C03635=1018.441,60.715,389.816,166.714,53.558,159.792
C03636=1018.447,60.965,389.800,166.716,53.550,159.791
C03637=1018.453,61.215,389.784,166.719,53.543,159.790
C03638=1018.458,61.464,389.769,166.722,53.536,159.789
C03639=1018.463,61.714,389.752,166.725,53.528,159.788
C03640=1018.469,61.964,389.737,166.727,53.521,159.787
C03641=1018.474,62.213,389.720,166.730,53.514,159.786
C03642=1018.480,62.462,389.704,166.732,53.506,159.785
C03643=1018.485,62.712,389.689,166.735,53.499,159.784
C03644=1018.491,62.961,389.673,166.738,53.491,159.784
C03645=1018.496,63.211,389.657,166.740,53.485,159.783
C03646=1018.502,63.460,389.641,166.743,53.477,159.782
C03647=1018.507,63.701,389.624,166.745,53.470,159.781
C03648=1018.512,63.942,389.609,166.748,53.463,159.780
C03649=1018.518,64.183,389.593,166.750,53.456,159.779
C03650=1018.523,64.424,389.578,166.753,53.449,159.779
C03651=1018.528,64.666,389.562,166.756,53.442,159.778
C03652=1018.533,64.907,389.546,166.758,53.435,159.777
C03653=1018.539,65.148,389.531,166.761,53.428,159.776
C03654=1018.543,65.389,389.515,166.763,53.421,159.775
C03655=1018.549,65.638,389.499,166.766,53.414,159.774
C03656=1018.554,65.888,389.482,166.768,53.407,159.773
C03657=1018.560,66.137,389.466,166.770,53.399,159.772
C03658=1018.565,66.387,389.450,166.773,53.392,159.772
C03659=1018.571,66.636,389.434,166.777,53.385,159.771
C03660=1018.576,66.885,389.418,166.778,53.378,159.770
C03661=1018.581,67.135,389.401,166.781,53.371,159.769
C03662=1018.587,67.384,389.385,166.785,53.363,159.768
C03663=1018.592,67.634,389.369,166.786,53.356,159.767
C03664=1018.597,67.883,389.353,166.789,53.349,159.766
C03665=1018.603,68.133,389.336,166.792,53.342,159.766
C03666=1018.609,68.382,389.320,166.795,53.334,159.765
C03667=1018.614,68.632,389.303,166.797,53.327,159.764
C03668=1018.619,68.880,389.287,166.800,53.320,159.763
C03669=1018.624,69.130,389.270,166.803,53.312,159.762
C03670=1018.630,69.380,389.253,166.805,53.306,159.761
C03671=1018.635,69.629,389.237,166.808,53.298,159.761
C03672=1018.640,69.878,389.221,166.811,53.291,159.760
C03673=1018.646,70.127,389.204,166.813,53.284,159.759
C03674=1018.651,70.377,389.187,166.816,53.277,159.758
C03675=1018.656,70.627,389.171,166.818,53.269,159.757
C03676=1018.662,70.876,389.154,166.820,53.262,159.756
C03677=1018.667,71.125,389.138,166.823,53.255,159.755
C03678=1018.673,71.374,389.122,166.826,53.248,159.755
C03679=1018.678,71.624,389.105,166.828,53.241,159.754
C03680=1018.683,71.874,389.088,166.831,53.234,159.753
C03681=1018.689,72.123,389.072,166.834,53.226,159.752
C03682=1018.694,72.372,389.055,166.836,53.219,159.751
C03683=1018.699,72.621,389.038,166.839,53.212,159.750
C03684=1018.705,72.871,389.022,166.842,53.205,159.749
C03685=1018.710,73.120,389.005,166.845,53.198,159.749
C03686=1018.716,73.370,388.988,166.847,53.190,159.747
C03687=1018.721,73.619,388.972,166.850,53.183,159.747
C03688=1018.726,73.868,388.956,166.853,53.176,159.746
C03689=1018.732,74.118,388.939,166.855,53.169,159.745
C03690=1018.737,74.367,388.922,166.858,53.162,159.744
C03691=1018.743,74.666,388.902,166.861,53.153,159.743
C03692=1018.750,74.965,388.882,166.864,53.144,159.742
C03693=1018.756,75.265,388.862,166.868,53.136,159.741
C03694=1018.763,75.563,388.842,166.871,53.127,159.740
C03695=1018.768,75.813,388.825,166.873,53.120,159.739
C03696=1018.774,76.062,388.809,166.876,53.112,159.738
C03697=1018.780,76.312,388.792,166.879,53.105,159.737
C03698=1018.785,76.560,388.775,166.881,53.098,159.736
C03699=1018.790,76.810,388.758,166.884,53.091,159.736
C03700=1018.796,77.059,388.742,166.887,53.084,159.735
C03701=1018.801,77.309,388.725,166.888,53.076,159.734
C03702=1018.806,77.559,388.708,166.891,53.069,159.733
C03703=1018.812,77.808,388.691,166.894,53.062,159.732
C03704=1018.817,78.057,388.674,166.897,53.055,159.731
C03705=1018.822,78.307,388.657,166.900,53.048,159.730
C03706=1018.828,78.556,388.640,166.903,53.041,159.730
C03707=1018.832,78.805,388.623,166.905,53.034,159.729
C03708=1018.837,79.055,388.606,166.908,53.027,159.728
C03709=1018.843,79.304,388.589,166.910,53.019,159.727
C03710=1018.848,79.553,388.572,166.912,53.012,159.726
C03711=1018.854,79.803,388.556,166.915,53.005,159.725
C03712=1018.860,80.052,388.538,166.919,52.998,159.725
C03713=1018.865,80.301,388.521,166.921,52.991,159.724
C03714=1018.870,80.551,388.504,166.924,52.984,159.723
C03715=1018.876,80.800,388.487,166.927,52.977,159.722
C03716=1018.881,81.050,388.470,166.928,52.969,159.721
C03717=1018.886,81.299,388.453,166.931,52.962,159.720
C03718=1018.891,81.548,388.436,166.934,52.955,159.719
C03719=1018.896,81.797,388.419,166.937,52.948,159.718
C03720=1018.902,82.046,388.401,166.940,52.941,159.718
C03721=1018.907,82.296,388.385,166.942,52.933,159.717
C03722=1018.912,82.546,388.368,166.944,52.927,159.716
C03723=1018.918,82.795,388.350,166.947,52.919,159.715
C03724=1018.923,83.044,388.333,166.950,52.912,159.714
C03725=1018.928,83.293,388.316,166.953,52.905,159.713
C03726=1018.934,83.543,388.299,166.955,52.898,159.712
C03727=1018.939,83.792,388.283,166.958,52.890,159.712
C03728=1018.945,84.041,388.265,166.961,52.883,159.711
C03729=1018.950,84.291,388.248,166.963,52.877,159.710
C03730=1018.956,84.540,388.231,166.966,52.869,159.709
C03731=1018.961,84.790,388.214,166.969,52.862,159.708
C03732=1018.966,85.039,388.196,166.971,52.855,159.707
C03733=1018.972,85.289,388.179,166.974,52.848,159.706
C03734=1018.977,85.538,388.162,166.977,52.840,159.705
C03735=1018.982,85.787,388.145,166.980,52.833,159.705
C03736=1018.988,86.036,388.127,166.982,52.826,159.704
C03737=1018.993,86.286,388.110,166.985,52.819,159.703
C03738=1018.998,86.536,388.094,166.988,52.811,159.702
C03739=1019.004,86.785,388.076,166.990,52.804,159.701
C03740=1019.009,87.034,388.059,166.993,52.797,159.700
C03741=1019.015,87.283,388.042,166.996,52.789,159.699
C03742=1019.020,87.532,388.024,166.999,52.782,159.698
C03743=1019.025,87.782,388.007,167.001,52.775,159.698
C03744=1019.032,88.031,387.990,167.004,52.768,159.697
C03745=1019.037,88.280,387.973,167.007,52.760,159.696
C03746=1019.042,88.529,387.956,167.010,52.753,159.695
C03747=1019.048,88.779,387.939,167.012,52.747,159.694
C03748=1019.053,89.028,387.921,167.015,52.739,159.693
C03749=1019.058,89.278,387.904,167.018,52.732,159.692
C03750=1019.064,89.528,387.886,167.021,52.725,159.692
C03751=1019.069,89.777,387.868,167.023,52.718,159.691
C03752=1019.074,90.027,387.852,167.026,52.711,159.690
C03753=1019.079,90.276,387.833,167.029,52.703,159.689
C03754=1019.085,90.525,387.816,167.031,52.696,159.688
C03755=1019.091,90.807,387.796,167.034,52.688,159.687
C03756=1019.097,91.090,387.776,167.037,52.680,159.686
C03757=1019.102,91.373,387.756,167.040,52.672,159.685
C03758=1019.108,91.654,387.737,167.044,52.664,159.684
C03759=1019.115,91.904,387.719,167.047,52.657,159.683
C03760=1019.119,92.154,387.701,167.048,52.650,159.682
C03761=1019.125,92.403,387.683,167.051,52.642,159.682
C03762=1019.130,92.652,387.667,167.055,52.635,159.681
C03763=1019.135,92.902,387.648,167.057,52.629,159.680
C03764=1019.140,93.151,387.631,167.060,52.622,159.679
C03765=1019.146,93.400,387.613,167.063,52.614,159.678
C03766=1019.151,93.649,387.596,167.065,52.607,159.677
C03767=1019.156,93.899,387.578,167.068,52.600,159.676
C03768=1019.161,94.148,387.561,167.071,52.593,159.676
C03769=1019.167,94.397,387.543,167.074,52.585,159.675
C03770=1019.173,94.646,387.525,167.076,52.578,159.674
C03771=1019.178,94.896,387.507,167.079,52.571,159.673
C03772=1019.183,95.145,387.490,167.082,52.564,159.672
C03773=1019.188,95.395,387.473,167.084,52.557,159.671
C03774=1019.194,95.644,387.455,167.087,52.550,159.670
C03775=1019.199,95.893,387.437,167.090,52.542,159.669
C03776=1019.204,96.142,387.419,167.093,52.535,159.669
C03777=1019.210,96.392,387.401,167.095,52.528,159.668
C03778=1019.215,96.641,387.383,167.098,52.521,159.667
C03779=1019.221,96.890,387.366,167.101,52.514,159.666
C03780=1019.226,97.140,387.349,167.104,52.507,159.665
C03781=1019.231,97.389,387.331,167.106,52.499,159.664
C03782=1019.236,97.638,387.313,167.109,52.492,159.663
C03783=1019.242,97.888,387.295,167.112,52.485,159.663
C03784=1019.248,98.137,387.278,167.115,52.477,159.662
C03785=1019.253,98.386,387.260,167.117,52.471,159.661
C03786=1019.258,98.635,387.242,167.120,52.464,159.660
C03787=1019.264,98.884,387.224,167.123,52.456,159.659
C03788=1019.270,99.134,387.206,167.126,52.449,159.658
C03789=1019.275,99.383,387.188,167.128,52.442,159.657
C03790=1019.280,99.632,387.171,167.131,52.435,159.656
C03791=1019.285,99.882,387.152,167.135,52.428,159.656
C03792=1019.290,100.131,387.135,167.137,52.421,159.655
C03793=1019.296,100.381,387.116,167.139,52.413,159.654
C03794=1019.301,100.630,387.098,167.143,52.406,159.653
C03795=1019.306,100.879,387.081,167.145,52.400,159.652
C03796=1019.311,101.129,387.062,167.148,52.393,159.651
C03797=1019.316,101.378,387.045,167.151,52.385,159.651
C03798=1019.322,101.627,387.026,167.153,52.378,159.649
C03799=1019.328,101.876,387.008,167.156,52.371,159.649
C03800=1019.332,102.126,386.990,167.159,52.364,159.648
C03801=1019.337,102.375,386.972,167.162,52.357,159.647
C03802=1019.343,102.625,386.954,167.164,52.350,159.646
C03803=1019.348,102.874,386.936,167.168,52.343,159.645
C03804=1019.354,103.123,386.918,167.170,52.335,159.644
C03805=1019.359,103.372,386.899,167.172,52.329,159.643
C03806=1019.365,103.621,386.881,167.176,52.322,159.643
C03807=1019.370,103.871,386.863,167.179,52.315,159.642
C03808=1019.374,104.120,386.845,167.182,52.307,159.641
C03809=1019.380,104.369,386.827,167.184,52.300,159.640
C03810=1019.385,104.619,386.809,167.187,52.293,159.639
C03811=1019.391,104.868,386.791,167.190,52.286,159.638
C03812=1019.396,105.117,386.772,167.192,52.279,159.637
C03813=1019.401,105.366,386.755,167.195,52.272,159.637
C03814=1019.407,105.616,386.736,167.198,52.264,159.636
C03815=1019.412,105.865,386.717,167.201,52.257,159.635
C03816=1019.417,106.114,386.700,167.203,52.250,159.634
C03817=1019.423,106.364,386.681,167.206,52.243,159.633
C03818=1019.428,106.613,386.664,167.209,52.236,159.632
C03819=1019.434,106.895,386.643,167.212,52.228,159.631
C03820=1019.441,107.178,386.622,167.216,52.219,159.630
C03821=1019.447,107.461,386.602,167.219,52.211,159.629
C03822=1019.453,107.743,386.581,167.222,52.204,159.628
C03823=1019.458,107.993,386.562,167.225,52.197,159.628
C03824=1019.463,108.242,386.544,167.228,52.189,159.627
C03825=1019.468,108.491,386.527,167.230,52.182,159.626
C03826=1019.474,108.741,386.507,167.234,52.175,159.625
C03827=1019.480,108.990,386.490,167.236,52.167,159.624
C03828=1019.484,109.239,386.472,167.239,52.160,159.623
C03829=1019.491,109.488,386.453,167.243,52.153,159.622
C03830=1019.495,109.737,386.435,167.245,52.147,159.622
C03831=1019.500,109.987,386.417,167.248,52.139,159.621
C03832=1019.506,110.236,386.397,167.251,52.132,159.620
C03833=1019.511,110.486,386.379,167.254,52.125,159.619
C03834=1019.517,110.734,386.361,167.256,52.118,159.618
C03835=1019.522,110.984,386.342,167.259,52.110,159.617
C03836=1019.527,111.233,386.324,167.262,52.103,159.616
C03837=1019.532,111.482,386.305,167.265,52.096,159.616
C03838=1019.538,111.732,386.287,167.268,52.090,159.615
C03839=1019.543,111.981,386.269,167.270,52.082,159.614
C03840=1019.548,112.231,386.250,167.274,52.075,159.613
C03841=1019.553,112.479,386.231,167.277,52.068,159.612
C03842=1019.558,112.729,386.213,167.279,52.061,159.611
C03843=1019.564,112.978,386.194,167.282,52.054,159.610
C03844=1019.569,113.227,386.175,167.285,52.047,159.610
C03845=1019.574,113.477,386.156,167.288,52.041,159.609
C03846=1019.580,113.726,386.137,167.291,52.034,159.608
C03847=1019.585,113.974,386.119,167.294,52.027,159.607
C03848=1019.590,114.224,386.100,167.296,52.019,159.606
C03849=1019.595,114.473,386.081,167.299,52.012,159.605
C03850=1019.600,114.722,386.062,167.302,52.005,159.605
C03851=1019.606,114.972,386.044,167.305,51.999,159.604
C03852=1019.611,115.221,386.025,167.308,51.992,159.603
C03853=1019.616,115.470,386.005,167.311,51.985,159.602
C03854=1019.620,115.720,385.987,167.314,51.978,159.601
C03855=1019.625,115.968,385.968,167.316,51.971,159.600
C03856=1019.631,116.218,385.949,167.319,51.963,159.599
C03857=1019.636,116.467,385.931,167.322,51.956,159.599
C03858=1019.642,116.717,385.911,167.325,51.950,159.598
C03859=1019.647,116.965,385.893,167.328,51.943,159.597
C03860=1019.652,117.215,385.874,167.331,51.936,159.596
C03861=1019.657,117.464,385.855,167.334,51.929,159.595
C03862=1019.663,117.714,385.836,167.336,51.921,159.594
C03863=1019.668,117.962,385.817,167.339,51.914,159.594
C03864=1019.673,118.212,385.799,167.343,51.907,159.593
C03865=1019.678,118.461,385.780,167.346,51.900,159.592
C03866=1019.683,118.710,385.761,167.348,51.894,159.591
C03867=1019.689,118.959,385.741,167.351,51.887,159.590
C03868=1019.694,119.209,385.723,167.354,51.879,159.589
C03869=1019.699,119.458,385.703,167.357,51.872,159.589
C03870=1019.704,119.707,385.685,167.360,51.865,159.588
C03871=1019.710,119.957,385.665,167.363,51.858,159.587
C03872=1019.715,120.205,385.646,167.366,51.851,159.586
C03873=1019.720,120.455,385.628,167.369,51.844,159.585
C03874=1019.725,120.704,385.609,167.372,51.837,159.584
C03875=1019.731,120.954,385.590,167.374,51.830,159.583
C03876=1019.736,121.202,385.571,167.378,51.823,159.583
C03877=1019.742,121.452,385.552,167.381,51.815,159.582
C03878=1019.747,121.700,385.533,167.384,51.808,159.581
C03879=1019.752,121.950,385.514,167.387,51.801,159.580
C03880=1019.757,122.199,385.495,167.389,51.795,159.579
C03881=1019.763,122.449,385.476,167.393,51.788,159.578
C03882=1019.768,122.697,385.457,167.395,51.780,159.577
C03883=1019.774,122.980,385.435,167.399,51.772,159.577
C03884=1019.780,123.263,385.413,167.402,51.764,159.576
C03885=1019.786,123.545,385.392,167.406,51.756,159.575
C03886=1019.792,123.828,385.370,167.408,51.748,159.574
C03887=1019.798,124.078,385.351,167.412,51.741,159.573
C03888=1019.803,124.326,385.332,167.415,51.734,159.572
C03889=1019.808,124.576,385.313,167.418,51.727,159.571
C03890=1019.814,124.824,385.294,167.421,51.719,159.570
C03891=1019.819,125.074,385.276,167.424,51.713,159.569
C03892=1019.824,125.323,385.257,167.427,51.706,159.569
C03893=1019.830,125.573,385.238,167.430,51.698,159.568
C03894=1019.835,125.822,385.218,167.433,51.691,159.567
C03895=1019.840,126.071,385.199,167.436,51.684,159.566
C03896=1019.845,126.321,385.180,167.439,51.677,159.565
C03897=1019.850,126.569,385.161,167.442,51.670,159.564
C03898=1019.856,126.819,385.141,167.445,51.663,159.563
C03899=1019.862,127.068,385.122,167.449,51.656,159.563
C03900=1019.867,127.317,385.103,167.451,51.648,159.562
C03901=1019.873,127.566,385.084,167.454,51.642,159.561
C03902=1019.878,127.816,385.065,167.457,51.635,159.560
C03903=1019.883,128.064,385.046,167.460,51.627,159.559
C03904=1019.889,128.314,385.027,167.463,51.620,159.558
C03905=1019.894,128.564,385.007,167.467,51.613,159.557
C03906=1019.899,128.812,384.988,167.469,51.605,159.557
C03907=1019.905,129.062,384.969,167.473,51.598,159.556
C03908=1019.910,129.311,384.950,167.476,51.592,159.555
C03909=1019.916,129.560,384.931,167.479,51.584,159.554
C03910=1019.921,129.809,384.911,167.482,51.577,159.553
C03911=1019.927,130.059,384.892,167.485,51.570,159.552
C03912=1019.932,130.307,384.872,167.488,51.563,159.552
C03913=1019.937,130.557,384.853,167.491,51.556,159.551
C03914=1019.942,130.806,384.833,167.494,51.549,159.550
C03915=1019.947,131.055,384.814,167.497,51.542,159.549
C03916=1019.952,131.305,384.794,167.500,51.535,159.548
C03917=1019.958,131.554,384.774,167.503,51.528,159.547
C03918=1019.963,131.803,384.755,167.506,51.521,159.547
C03919=1019.968,132.052,384.736,167.509,51.514,159.546
C03920=1019.974,132.301,384.716,167.512,51.507,159.545
C03921=1019.979,132.550,384.696,167.516,51.500,159.544
C03922=1019.984,132.799,384.677,167.519,51.493,159.543
C03923=1019.989,133.049,384.657,167.521,51.486,159.542
C03924=1019.995,133.297,384.637,167.524,51.479,159.541
C03925=1020.000,133.547,384.618,167.527,51.472,159.541
C03926=1020.005,133.797,384.598,167.531,51.465,159.540
C03927=1020.011,134.045,384.578,167.534,51.458,159.539
C03928=1020.016,134.294,384.559,167.537,51.451,159.538
C03929=1020.021,134.544,384.540,167.540,51.443,159.537
C03930=1020.027,134.793,384.519,167.543,51.437,159.536
C03931=1020.032,135.042,384.500,167.546,51.430,159.536
C03932=1020.037,135.291,384.480,167.549,51.423,159.535
C03933=1020.043,135.540,384.460,167.553,51.416,159.534
C03934=1020.048,135.790,384.441,167.555,51.409,159.533
C03935=1020.053,136.039,384.422,167.559,51.402,159.532
C03936=1020.058,136.288,384.401,167.562,51.395,159.531
C03937=1020.064,136.537,384.382,167.565,51.388,159.531
C03938=1020.069,136.786,384.361,167.569,51.381,159.530
C03939=1020.074,137.035,384.342,167.571,51.374,159.529
C03940=1020.079,137.284,384.322,167.574,51.367,159.528
C03941=1020.085,137.534,384.303,167.577,51.360,159.527
C03942=1020.090,137.783,384.282,167.581,51.353,159.527
C03943=1020.096,138.032,384.263,167.584,51.346,159.526
C03944=1020.100,138.281,384.243,167.587,51.338,159.525
C03945=1020.105,138.530,384.223,167.590,51.331,159.524
C03946=1020.111,138.780,384.202,167.593,51.325,159.523
C03947=1020.117,139.062,384.180,167.596,51.317,159.522
C03948=1020.123,139.345,384.158,167.600,51.309,159.521
C03949=1020.129,139.627,384.135,167.604,51.301,159.520
C03950=1020.135,139.910,384.112,167.607,51.293,159.519
C03951=1020.140,140.158,384.093,167.611,51.287,159.519
C03952=1020.145,140.408,384.072,167.614,51.280,159.518
C03953=1020.150,140.657,384.052,167.617,51.273,159.517
C03954=1020.155,140.906,384.032,167.620,51.265,159.516
C03955=1020.161,141.155,384.012,167.624,51.258,159.515
C03956=1020.166,141.404,383.992,167.627,51.251,159.515
C03957=1020.171,141.653,383.972,167.630,51.245,159.514
C03958=1020.177,141.902,383.952,167.634,51.238,159.513
C03959=1020.182,142.152,383.932,167.636,51.231,159.512
C03960=1020.187,142.401,383.912,167.639,51.224,159.511
C03961=1020.192,142.650,383.891,167.642,51.217,159.510
C03962=1020.197,142.899,383.872,167.646,51.210,159.510
C03963=1020.203,143.148,383.852,167.649,51.203,159.509
C03964=1020.208,143.397,383.831,167.652,51.196,159.508
C03965=1020.214,143.646,383.811,167.656,51.189,159.507
C03966=1020.219,143.896,383.791,167.659,51.182,159.506
C03967=1020.224,144.145,383.771,167.662,51.175,159.506
C03968=1020.229,144.394,383.750,167.665,51.168,159.505
C03969=1020.235,144.643,383.731,167.669,51.161,159.504
C03970=1020.240,144.893,383.710,167.672,51.154,159.503
C03971=1020.245,145.141,383.690,167.675,51.147,159.502
C03972=1020.251,145.390,383.670,167.678,51.140,159.501
C03973=1020.256,145.640,383.650,167.682,51.133,159.501
C03974=1020.261,145.889,383.630,167.685,51.126,159.500
C03975=1020.266,146.138,383.609,167.688,51.119,159.499
C03976=1020.272,146.387,383.589,167.692,51.112,159.498
C03977=1020.277,146.636,383.568,167.695,51.105,159.498
C03978=1020.282,146.885,383.548,167.697,51.099,159.497
C03979=1020.288,147.134,383.528,167.700,51.091,159.496
C03980=1020.293,147.384,383.508,167.704,51.084,159.495
C03981=1020.298,147.633,383.487,167.707,51.077,159.494
C03982=1020.304,147.882,383.467,167.710,51.071,159.493
C03983=1020.309,148.131,383.446,167.714,51.064,159.493
C03984=1020.314,148.379,383.426,167.717,51.057,159.492
C03985=1020.319,148.629,383.405,167.721,51.050,159.491
C03986=1020.324,148.878,383.385,167.724,51.043,159.490
C03987=1020.329,149.127,383.364,167.727,51.036,159.489
C03988=1020.335,149.376,383.344,167.731,51.029,159.489
C03989=1020.340,149.625,383.323,167.734,51.022,159.488
C03990=1020.345,149.874,383.303,167.737,51.016,159.487
C03991=1020.350,150.123,383.282,167.740,51.008,159.486
C03992=1020.356,150.372,383.261,167.744,51.001,159.485
C03993=1020.361,150.622,383.241,167.747,50.994,159.485
C03994=1020.366,150.871,383.220,167.751,50.988,159.484
C03995=1020.371,151.120,383.200,167.754,50.981,159.483
C03996=1020.377,151.369,383.179,167.757,50.974,159.482
C03997=1020.382,151.618,383.159,167.761,50.967,159.481
C03998=1020.387,151.867,383.138,167.764,50.960,159.481
C03999=1020.392,152.116,383.118,167.767,50.953,159.480
C04000=1020.398,152.365,383.097,167.771,50.946,159.479
C04001=1020.403,152.614,383.076,167.774,50.939,159.478
C04002=1020.408,152.863,383.055,167.777,50.932,159.477
C04003=1020.414,153.112,383.035,167.781,50.925,159.477
C04004=1020.419,153.361,383.014,167.784,50.918,159.476
C04005=1020.424,153.610,382.994,167.787,50.912,159.475
C04006=1020.429,153.860,382.972,167.791,50.905,159.474
C04007=1020.434,154.109,382.952,167.794,50.898,159.473
C04008=1020.440,154.358,382.930,167.798,50.891,159.473
C04009=1020.445,154.607,382.910,167.801,50.884,159.472
C04010=1020.451,154.857,382.889,167.804,50.877,159.471
C04011=1020.456,155.139,382.865,167.807,50.870,159.470
C04012=1020.462,155.421,382.842,167.811,50.862,159.469
C04013=1020.469,155.703,382.818,167.815,50.854,159.468
C04014=1020.474,155.985,382.795,167.819,50.846,159.467
C04015=1020.480,156.234,382.774,167.823,50.839,159.467
C04016=1020.484,156.483,382.753,167.826,50.833,159.466
C04017=1020.490,156.733,382.732,167.830,50.826,159.465
C04018=1020.495,156.982,382.711,167.833,50.819,159.464
C04019=1020.501,157.231,382.690,167.837,50.812,159.464
C04020=1020.506,157.480,382.670,167.840,50.805,159.463
C04021=1020.511,157.729,382.649,167.843,50.799,159.462
C04022=1020.516,157.978,382.627,167.847,50.792,159.461
C04023=1020.521,158.227,382.607,167.850,50.785,159.460
C04024=1020.527,158.476,382.586,167.853,50.777,159.459
C04025=1020.532,158.725,382.565,167.857,50.771,159.459
C04026=1020.538,158.974,382.544,167.860,50.764,159.458
C04027=1020.543,159.223,382.522,167.864,50.758,159.457
C04028=1020.547,159.473,382.501,167.867,50.751,159.457
C04029=1020.553,159.721,382.480,167.871,50.744,159.456
C04030=1020.558,159.971,382.458,167.874,50.737,159.455
C04031=1020.563,160.219,382.437,167.877,50.730,159.454
C04032=1020.568,160.468,382.415,167.881,50.724,159.453
C04033=1020.572,160.717,382.394,167.885,50.717,159.453
C04034=1020.579,160.967,382.372,167.888,50.711,159.452
C04035=1020.583,161.216,382.351,167.892,50.704,159.451
C04036=1020.588,161.465,382.329,167.895,50.697,159.451
C04037=1020.593,161.713,382.308,167.898,50.690,159.450
C04038=1020.598,161.963,382.287,167.902,50.683,159.449
C04039=1020.604,162.211,382.266,167.906,50.677,159.448
C04040=1020.608,162.460,382.244,167.909,50.671,159.448
C04041=1020.614,162.710,382.222,167.912,50.664,159.447
C04042=1020.619,162.959,382.201,167.916,50.657,159.446
C04043=1020.624,163.208,382.179,167.919,50.650,159.445
C04044=1020.628,163.457,382.158,167.923,50.643,159.444
C04045=1020.634,163.706,382.137,167.927,50.637,159.444
C04046=1020.639,163.954,382.115,167.930,50.630,159.443
C04047=1020.645,164.204,382.094,167.933,50.624,159.442
C04048=1020.649,164.453,382.072,167.937,50.617,159.442
C04049=1020.654,164.702,382.050,167.940,50.610,159.441
C04050=1020.660,164.950,382.029,167.944,50.603,159.440
C04051=1020.665,165.200,382.008,167.947,50.597,159.439
C04052=1020.670,165.449,381.986,167.951,50.590,159.439
C04053=1020.675,165.698,381.964,167.954,50.584,159.438
C04054=1020.680,165.947,381.943,167.958,50.577,159.437
C04055=1020.685,166.197,381.921,167.961,50.570,159.436
C04056=1020.691,166.445,381.900,167.965,50.563,159.435
C04057=1020.696,166.694,381.878,167.969,50.556,159.435
C04058=1020.701,166.943,381.857,167.973,50.549,159.434
C04059=1020.707,167.192,381.834,167.977,50.543,159.433
C04060=1020.711,167.441,381.813,167.980,50.537,159.433
C04061=1020.717,167.690,381.792,167.983,50.530,159.432
C04062=1020.722,167.939,381.770,167.987,50.523,159.431
C04063=1020.727,168.188,381.748,167.990,50.516,159.430
C04064=1020.733,168.437,381.727,167.994,50.509,159.430
C04065=1020.737,168.686,381.705,167.997,50.503,159.429
C04066=1020.743,168.936,381.683,168.001,50.496,159.428
C04067=1020.748,169.184,381.662,168.005,50.490,159.427
C04068=1020.753,169.433,381.640,168.009,50.483,159.427
C04069=1020.759,169.682,381.618,168.012,50.476,159.426
C04070=1020.764,169.931,381.597,168.016,50.469,159.425
C04071=1020.769,170.180,381.575,168.019,50.462,159.424
C04072=1020.775,170.429,381.553,168.023,50.456,159.424
C04073=1020.780,170.678,381.531,168.026,50.449,159.423
C04074=1020.785,170.927,381.509,168.030,50.442,159.422
C04075=1020.791,171.209,381.485,168.034,50.435,159.421
C04076=1020.797,171.491,381.460,168.038,50.427,159.420
C04077=1020.803,171.773,381.436,168.042,50.420,159.420
C04078=1020.809,172.055,381.411,168.047,50.412,159.419
C04079=1020.814,172.304,381.389,168.050,50.405,159.418
C04080=1020.819,172.553,381.368,168.055,50.399,159.417
C04081=1020.825,172.802,381.345,168.058,50.392,159.417
C04082=1020.830,173.051,381.324,168.062,50.385,159.416
C04083=1020.836,173.300,381.302,168.065,50.378,159.415
C04084=1020.841,173.549,381.280,168.069,50.372,159.414
C04085=1020.847,173.798,381.258,168.073,50.365,159.414
C04086=1020.851,174.047,381.236,168.077,50.358,159.413
C04087=1020.856,174.296,381.215,168.080,50.351,159.412
C04088=1020.862,174.545,381.193,168.084,50.344,159.411
C04089=1020.867,174.794,381.171,168.087,50.338,159.411
C04090=1020.873,175.043,381.149,168.092,50.331,159.410
C04091=1020.878,175.292,381.128,168.095,50.324,159.409
C04092=1020.884,175.541,381.105,168.099,50.318,159.408
C04093=1020.889,175.790,381.083,168.102,50.311,159.408
C04094=1020.895,176.039,381.061,168.107,50.304,159.407
C04095=1020.900,176.288,381.039,168.110,50.297,159.406
C04096=1020.905,176.537,381.017,168.114,50.290,159.405
C04097=1020.911,176.786,380.996,168.117,50.284,159.405
C04098=1020.916,177.035,380.974,168.122,50.277,159.404
C04099=1020.921,177.284,380.952,168.126,50.271,159.403
C04100=1020.928,177.532,380.929,168.129,50.264,159.402
C04101=1020.932,177.781,380.907,168.133,50.257,159.402
C04102=1020.938,178.031,380.885,168.137,50.250,159.401
C04103=1020.943,178.279,380.864,168.141,50.243,159.400
C04104=1020.949,178.529,380.842,168.144,50.237,159.399
C04105=1020.954,178.777,380.819,168.149,50.230,159.399
C04106=1020.960,179.026,380.798,168.153,50.223,159.398
C04107=1020.965,179.275,380.776,168.156,50.217,159.397
C04108=1020.970,179.525,380.753,168.161,50.210,159.397
C04109=1020.976,179.774,380.732,168.164,50.203,159.396
C04110=1020.982,180.022,380.709,168.168,50.196,159.395
C04111=1020.987,180.271,380.687,168.172,50.189,159.394
C04112=1020.993,180.520,380.666,168.176,50.183,159.394
C04113=1020.998,180.769,380.643,168.179,50.176,159.393
C04114=1021.004,181.018,380.621,168.183,50.169,159.392
C04115=1021.009,181.267,380.599,168.187,50.163,159.392
C04116=1021.015,181.516,380.577,168.191,50.156,159.391
C04117=1021.020,181.765,380.554,168.195,50.149,159.390
C04118=1021.025,182.014,380.532,168.199,50.142,159.389
C04119=1021.032,182.263,380.510,168.202,50.136,159.389
C04120=1021.036,182.512,380.487,168.206,50.130,159.388
C04121=1021.042,182.761,380.464,168.211,50.123,159.387
C04122=1021.046,183.011,380.442,168.215,50.116,159.387
C04123=1021.051,183.259,380.419,168.218,50.110,159.386
C04124=1021.057,183.508,380.396,168.222,50.103,159.385
C04125=1021.062,183.756,380.374,168.226,50.097,159.384
C04126=1021.067,184.006,380.351,168.230,50.090,159.384
C04127=1021.073,184.255,380.328,168.234,50.084,159.383
C04128=1021.077,184.503,380.306,168.238,50.077,159.382
C04129=1021.082,184.753,380.282,168.241,50.071,159.382
C04130=1021.088,185.002,380.259,168.245,50.065,159.381
C04131=1021.093,185.250,380.238,168.250,50.058,159.381
C04132=1021.098,185.500,380.214,168.253,50.052,159.380
C04133=1021.103,185.748,380.191,168.257,50.045,159.379
C04134=1021.109,185.997,380.168,168.261,50.039,159.378
C04135=1021.114,186.246,380.146,168.265,50.032,159.378
C04136=1021.119,186.495,380.123,168.269,50.026,159.377
C04137=1021.124,186.744,380.100,168.273,50.019,159.376
C04138=1021.129,186.993,380.077,168.278,50.013,159.376
C04139=1021.135,187.274,380.051,168.282,50.005,159.375
C04140=1021.142,187.556,380.026,168.286,49.998,159.374
C04141=1021.148,187.837,380.000,168.291,49.991,159.374
C04142=1021.154,188.119,379.974,168.295,49.983,159.373
C04143=1021.158,188.368,379.951,168.299,49.977,159.372
C04144=1021.164,188.617,379.928,168.304,49.970,159.371
C04145=1021.169,188.866,379.905,168.307,49.964,159.371
C04146=1021.174,189.114,379.882,168.311,49.958,159.370
C04147=1021.180,189.363,379.859,168.316,49.951,159.369
C04148=1021.185,189.612,379.836,168.319,49.945,159.369
C04149=1021.190,189.861,379.812,168.323,49.938,159.368
C04150=1021.195,190.110,379.790,168.328,49.932,159.367
C04151=1021.201,190.359,379.767,168.331,49.925,159.367
C04152=1021.206,190.608,379.744,168.335,49.919,159.366
C04153=1021.212,190.857,379.721,168.340,49.912,159.365
C04154=1021.217,191.105,379.698,168.344,49.906,159.365
C04155=1021.222,191.354,379.675,168.347,49.900,159.364
C04156=1021.227,191.603,379.652,168.352,49.893,159.363
C04157=1021.233,191.852,379.629,168.356,49.887,159.363
C04158=1021.238,192.101,379.605,168.360,49.881,159.362
C04159=1021.244,192.350,379.582,168.364,49.874,159.361
C04160=1021.249,192.598,379.560,168.368,49.867,159.361
C04161=1021.254,192.848,379.536,168.373,49.861,159.360
C04162=1021.260,193.097,379.513,168.376,49.854,159.359
C04163=1021.265,193.345,379.490,168.380,49.848,159.359
C04164=1021.270,193.595,379.467,168.385,49.841,159.358
C04165=1021.276,193.844,379.444,168.389,49.835,159.357
C04166=1021.281,194.092,379.421,168.393,49.828,159.357
C04167=1021.286,194.341,379.398,168.397,49.822,159.356
C04168=1021.292,194.589,379.374,168.401,49.815,159.355
C04169=1021.298,194.838,379.351,168.406,49.809,159.355
C04170=1021.303,195.087,379.328,168.409,49.802,159.354
C04171=1021.309,195.336,379.305,168.414,49.796,159.353
C04172=1021.314,195.585,379.282,168.418,49.790,159.353
C04173=1021.319,195.834,379.258,168.423,49.783,159.352
C04174=1021.325,196.083,379.235,168.426,49.777,159.351
C04175=1021.330,196.332,379.212,168.431,49.770,159.351
C04176=1021.336,196.580,379.188,168.435,49.764,159.350
C04177=1021.341,196.829,379.165,168.439,49.758,159.350
C04178=1021.346,197.078,379.142,168.443,49.751,159.349
C04179=1021.352,197.327,379.119,168.447,49.745,159.348
C04180=1021.358,197.576,379.096,168.452,49.738,159.348
C04181=1021.363,197.825,379.072,168.456,49.732,159.347
C04182=1021.369,198.073,379.049,168.460,49.725,159.346
C04183=1021.375,198.322,379.026,168.464,49.719,159.346
C04184=1021.380,198.572,379.002,168.469,49.712,159.345
C04185=1021.386,198.820,378.979,168.473,49.706,159.344
C04186=1021.391,199.069,378.956,168.477,49.699,159.344
C04187=1021.396,199.318,378.932,168.481,49.693,159.343
C04188=1021.402,199.566,378.909,168.486,49.687,159.342
C04189=1021.407,199.815,378.885,168.490,49.680,159.342
C04190=1021.412,200.065,378.861,168.495,49.674,159.341
C04191=1021.418,200.313,378.838,168.498,49.668,159.341
C04192=1021.423,200.562,378.814,168.503,49.661,159.340
C04193=1021.429,200.811,378.790,168.507,49.655,159.339
C04194=1021.434,201.060,378.766,168.512,49.649,159.339
C04195=1021.440,201.308,378.743,168.516,49.642,159.338
C04196=1021.445,201.557,378.719,168.520,49.636,159.337
C04197=1021.450,201.806,378.695,168.524,49.630,159.337
C04198=1021.456,202.054,378.671,168.529,49.624,159.336
C04199=1021.461,202.303,378.648,168.533,49.617,159.336
C04200=1021.467,202.553,378.623,168.538,49.611,159.335
C04201=1021.472,202.802,378.600,168.542,49.605,159.334
C04202=1021.478,203.050,378.576,168.547,49.599,159.334
C04203=1021.506,204.302,378.455,168.985,49.689,159.423
C04204=1021.511,204.516,378.432,168.988,49.684,159.422
C04205=1021.516,204.731,378.411,168.992,49.680,159.422
C04206=1021.522,204.946,378.389,168.994,49.676,159.421
C04207=1021.528,205.161,378.367,168.998,49.671,159.421
C04208=1021.533,205.376,378.345,169.001,49.666,159.420
C04209=1021.538,205.591,378.323,169.003,49.662,159.420
C04210=1021.543,205.805,378.301,169.007,49.657,159.419
C04211=1021.550,206.055,378.275,169.010,49.652,159.419
C04212=1021.556,206.303,378.250,169.014,49.646,159.418
C04213=1021.563,206.552,378.225,169.017,49.641,159.418
C04214=1021.569,206.800,378.199,169.020,49.636,159.417
C04215=1021.575,207.049,378.173,169.024,49.630,159.417
C04216=1021.582,207.297,378.148,169.027,49.625,159.416
C04217=1021.588,207.546,378.123,169.031,49.620,159.415
C04218=1021.594,207.795,378.097,169.035,49.614,159.415
C04219=1021.601,208.043,378.071,169.038,49.609,159.414
C04220=1021.606,208.292,378.045,169.041,49.605,159.414
C04221=1021.612,208.540,378.020,169.044,49.599,159.413
C04222=1021.619,208.789,377.994,169.048,49.594,159.413
C04223=1021.626,209.038,377.968,169.051,49.589,159.412
C04224=1021.632,209.287,377.943,169.055,49.584,159.412
C04225=1021.638,209.535,377.918,169.059,49.579,159.411
C04226=1021.644,209.783,377.891,169.062,49.573,159.410
C04227=1021.650,210.032,377.866,169.065,49.568,159.410
C04228=1021.656,210.280,377.840,169.069,49.563,159.409
C04229=1021.663,210.529,377.814,169.073,49.558,159.409
C04230=1021.669,210.778,377.789,169.076,49.553,159.408
C04231=1021.675,211.027,377.762,169.079,49.548,159.408
C04232=1021.681,211.275,377.736,169.083,49.543,159.407
C04233=1021.688,211.523,377.710,169.087,49.538,159.407
C04234=1021.693,211.772,377.684,169.090,49.532,159.406
C04235=1021.700,212.020,377.658,169.094,49.527,159.406
C04236=1021.706,212.269,377.633,169.097,49.522,159.405
C04237=1021.712,212.517,377.606,169.100,49.517,159.404
C04238=1021.719,212.767,377.581,169.104,49.512,159.404
C04239=1021.725,213.015,377.555,169.108,49.507,159.404
C04240=1021.731,213.264,377.529,169.111,49.502,159.403
C04241=1021.737,213.512,377.503,169.114,49.497,159.402
C04242=1021.743,213.761,377.477,169.118,49.492,159.402
C04243=1021.750,214.010,377.450,169.122,49.487,159.401
C04244=1021.756,214.258,377.425,169.125,49.482,159.401
C04245=1021.763,214.506,377.399,169.128,49.477,159.400
C04246=1021.768,214.755,377.372,169.133,49.472,159.400
C04247=1021.775,215.004,377.347,169.136,49.467,159.399
C04248=1021.782,215.252,377.321,169.139,49.462,159.399
C04249=1021.787,215.501,377.295,169.143,49.457,159.398
C04250=1021.794,215.749,377.269,169.147,49.452,159.398
C04251=1021.800,215.997,377.243,169.150,49.447,159.397
C04252=1021.806,216.247,377.216,169.153,49.442,159.397
C04253=1021.813,216.495,377.190,169.157,49.438,159.396
C04254=1021.819,216.743,377.164,169.161,49.433,159.396
C04255=1021.825,216.993,377.138,169.164,49.428,159.395
C04256=1021.832,217.241,377.112,169.168,49.423,159.395
C04257=1021.838,217.489,377.086,169.171,49.418,159.394
C04258=1021.844,217.738,377.060,169.175,49.413,159.394
C04259=1021.851,217.987,377.033,169.179,49.408,159.393
C04260=1021.857,218.235,377.007,169.182,49.403,159.393
C04261=1021.863,218.484,376.981,169.186,49.398,159.392
C04262=1021.869,218.732,376.955,169.190,49.394,159.392
C04263=1021.875,218.949,376.931,169.192,49.390,159.392
C04264=1021.880,219.166,376.909,169.196,49.385,159.391
C04265=1021.886,219.383,376.886,169.198,49.381,159.391
C04266=1021.891,219.600,376.863,169.202,49.377,159.390
C04267=1021.896,219.817,376.839,169.204,49.373,159.390
C04268=1021.901,220.034,376.817,169.208,49.369,159.389
C04269=1021.907,220.251,376.794,169.212,49.364,159.389
C04270=1021.913,220.468,376.770,169.214,49.361,159.389
C04271=1021.919,220.717,376.744,169.218,49.356,159.388
C04272=1021.925,220.965,376.717,169.222,49.351,159.388
C04273=1021.932,221.214,376.691,169.226,49.346,159.387
C04274=1021.937,221.462,376.664,169.229,49.341,159.387
C04275=1021.944,221.710,376.638,169.232,49.337,159.386
C04276=1021.950,221.959,376.611,169.236,49.332,159.386
C04277=1021.956,222.207,376.584,169.240,49.327,159.385
C04278=1021.963,222.456,376.558,169.244,49.323,159.385
C04279=1021.969,222.705,376.531,169.247,49.318,159.385
C04280=1021.975,222.953,376.505,169.250,49.313,159.384
C04281=1021.982,223.202,376.478,169.254,49.309,159.384
C04282=1021.988,223.450,376.452,169.258,49.304,159.383
C04283=1021.993,223.698,376.425,169.262,49.299,159.383
C04284=1022.001,223.947,376.399,169.265,49.294,159.382
C04285=1022.006,224.196,376.372,169.269,49.290,159.382
C04286=1022.013,224.445,376.345,169.272,49.285,159.381
C04287=1022.019,224.693,376.319,169.276,49.280,159.381
C04288=1022.026,224.942,376.292,169.280,49.276,159.381
C04289=1022.032,225.190,376.266,169.283,49.271,159.380
C04290=1022.038,225.438,376.239,169.287,49.267,159.380
C04291=1022.044,225.687,376.212,169.290,49.262,159.379
C04292=1022.051,225.935,376.185,169.295,49.257,159.379
C04293=1022.057,226.184,376.158,169.298,49.253,159.378
C04294=1022.063,226.432,376.132,169.302,49.248,159.378
C04295=1022.070,226.681,376.105,169.305,49.244,159.378
C04296=1022.076,226.929,376.079,169.309,49.239,159.377
C04297=1022.083,227.178,376.052,169.313,49.235,159.377
C04298=1022.089,227.426,376.024,169.317,49.230,159.376
C04299=1022.094,227.674,375.998,169.320,49.226,159.376
C04300=1022.101,227.923,375.971,169.324,49.221,159.376
C04301=1022.108,228.171,375.944,169.327,49.217,159.375
C04302=1022.114,228.420,375.917,169.331,49.212,159.375
C04303=1022.120,228.668,375.890,169.335,49.208,159.375
C04304=1022.126,228.917,375.863,169.339,49.203,159.374
C04305=1022.132,229.165,375.836,169.342,49.199,159.374
C04306=1022.139,229.414,375.809,169.346,49.195,159.373
C04307=1022.144,229.662,375.782,169.349,49.190,159.373
C04308=1022.151,229.911,375.754,169.353,49.186,159.372
C04309=1022.157,230.159,375.728,169.358,49.181,159.372
C04310=1022.164,230.407,375.701,169.361,49.177,159.372
C04311=1022.171,230.656,375.674,169.365,49.172,159.371
C04312=1022.176,230.905,375.646,169.368,49.168,159.371
C04313=1022.182,231.154,375.619,169.372,49.164,159.370
C04314=1022.188,231.402,375.592,169.375,49.159,159.370
C04315=1022.195,231.650,375.564,169.379,49.155,159.370
C04316=1022.200,231.899,375.538,169.382,49.150,159.369
C04317=1022.207,232.147,375.510,169.387,49.146,159.369
C04318=1022.213,232.396,375.483,169.391,49.142,159.369
C04319=1022.220,232.644,375.455,169.394,49.137,159.368
C04320=1022.225,232.892,375.429,169.398,49.133,159.368
C04321=1022.232,233.141,375.401,169.402,49.129,159.368
C04322=1022.239,233.389,375.373,169.405,49.125,159.367
C04323=1022.244,233.602,375.351,169.409,49.121,159.367
C04324=1022.249,233.815,375.327,169.412,49.117,159.367
C04325=1022.254,234.028,375.303,169.416,49.113,159.366
C04326=1022.260,234.241,375.280,169.419,49.110,159.366
C04327=1022.265,234.455,375.257,169.421,49.106,159.366
C04328=1022.271,234.667,375.233,169.425,49.103,159.365
C04329=1022.277,234.880,375.210,169.428,49.099,159.365
C04330=1022.281,235.093,375.186,169.432,49.095,159.365
C04331=1022.288,235.342,375.159,169.436,49.091,159.364
C04332=1022.294,235.590,375.132,169.439,49.087,159.364
C04333=1022.300,235.838,375.104,169.443,49.083,159.364
C04334=1022.307,236.087,375.077,169.446,49.078,159.363
C04335=1022.313,236.335,375.049,169.450,49.074,159.363
C04336=1022.320,236.584,375.022,169.454,49.070,159.363
C04337=1022.326,236.833,374.995,169.458,49.065,159.362
C04338=1022.332,237.080,374.967,169.462,49.061,159.362
C04339=1022.339,237.329,374.940,169.466,49.057,159.362
C04340=1022.345,237.578,374.911,169.469,49.053,159.361
C04341=1022.350,237.826,374.885,169.473,49.049,159.361
C04342=1022.357,238.074,374.857,169.477,49.045,159.361
C04343=1022.364,238.323,374.829,169.480,49.040,159.360
C04344=1022.370,238.571,374.802,169.484,49.036,159.360
C04345=1022.376,238.820,374.775,169.489,49.032,159.360
C04346=1022.383,239.068,374.747,169.492,49.028,159.359
C04347=1022.390,239.317,374.719,169.496,49.023,159.359
C04348=1022.395,239.565,374.691,169.500,49.020,159.359
C04349=1022.402,239.813,374.664,169.504,49.016,159.358
C04350=1022.408,240.061,374.636,169.507,49.011,159.358
C04351=1022.414,240.309,374.608,169.511,49.007,159.358
C04352=1022.420,240.558,374.580,169.515,49.004,159.358
C04353=1022.426,240.807,374.552,169.519,49.000,159.357
C04354=1022.433,241.055,374.524,169.523,48.995,159.357
C04355=1022.439,241.303,374.497,169.527,48.991,159.357
C04356=1022.445,241.552,374.468,169.531,48.987,159.356
C04357=1022.452,241.800,374.441,169.535,48.983,159.356
C04358=1022.458,242.049,374.412,169.538,48.979,159.356
C04359=1022.464,242.297,374.385,169.542,48.976,159.356
C04360=1022.470,242.545,374.357,169.546,48.971,159.355
C04361=1022.476,242.794,374.329,169.550,48.967,159.355
C04362=1022.483,243.042,374.301,169.554,48.964,159.355
C04363=1022.489,243.291,374.273,169.557,48.960,159.354
C04364=1022.495,243.539,374.246,169.561,48.955,159.354
C04365=1022.501,243.787,374.217,169.566,48.952,159.354
C04366=1022.508,244.035,374.189,169.570,48.947,159.353
C04367=1022.514,244.284,374.160,169.574,48.944,159.353
C04368=1022.519,244.532,374.132,169.577,48.940,159.353
C04369=1022.526,244.780,374.104,169.581,48.936,159.353
C04370=1022.532,245.029,374.076,169.585,48.932,159.352
C04371=1022.538,245.277,374.047,169.589,48.928,159.352
C04372=1022.545,245.525,374.019,169.593,48.924,159.352
C04373=1022.550,245.773,373.991,169.597,48.921,159.352
C04374=1022.556,246.022,373.963,169.600,48.917,159.351
C04375=1022.563,246.270,373.934,169.604,48.913,159.351
C04376=1022.569,246.519,373.906,169.608,48.910,159.351
C04377=1022.575,246.767,373.878,169.612,48.905,159.351
C04378=1022.582,247.015,373.849,169.616,48.902,159.351
C04379=1022.588,247.263,373.821,169.620,48.898,159.350
C04380=1022.594,247.512,373.793,169.624,48.894,159.350
C04381=1022.601,247.760,373.764,169.627,48.890,159.350
C04382=1022.607,248.009,373.736,169.631,48.887,159.349
C04383=1022.617,248.429,373.688,169.638,48.880,159.349
C04384=1022.627,248.848,373.640,169.645,48.874,159.349
C04385=1022.638,249.268,373.592,169.652,48.867,159.348
C04386=1022.649,249.688,373.544,169.659,48.861,159.348
C04387=1022.655,249.936,373.515,169.663,48.857,159.348
C04388=1022.662,250.184,373.487,169.667,48.854,159.348
C04389=1022.668,250.432,373.458,169.671,48.850,159.347
C04390=1022.674,250.681,373.430,169.674,48.846,159.347
C04391=1022.680,250.929,373.401,169.679,48.843,159.347
C04392=1022.687,251.178,373.373,169.683,48.839,159.347
C04393=1022.693,251.426,373.344,169.686,48.835,159.346
C04394=1022.699,251.674,373.316,169.690,48.831,159.346
C04395=1022.706,251.922,373.288,169.694,48.828,159.346
C04396=1022.712,252.170,373.259,169.698,48.824,159.346
C04397=1022.718,252.419,373.230,169.702,48.820,159.345
C04398=1022.725,252.667,373.201,169.706,48.817,159.345
C04399=1022.731,252.916,373.173,169.711,48.813,159.345
C04400=1022.738,253.164,373.144,169.715,48.810,159.345
C04401=1022.744,253.412,373.115,169.719,48.805,159.345
C04402=1022.751,253.660,373.087,169.723,48.802,159.344
C04403=1022.757,253.909,373.058,169.727,48.798,159.344
C04404=1022.763,254.157,373.029,169.731,48.795,159.344
C04405=1022.770,254.405,373.001,169.735,48.791,159.344
C04406=1022.776,254.653,372.972,169.739,48.788,159.344
C04407=1022.782,254.901,372.943,169.742,48.784,159.343
C04408=1022.789,255.149,372.915,169.746,48.780,159.343
C04409=1022.795,255.398,372.887,169.751,48.776,159.343
C04410=1022.801,255.646,372.858,169.755,48.773,159.343
C04411=1022.808,255.894,372.828,169.759,48.770,159.343
C04412=1022.815,256.143,372.800,169.763,48.766,159.343
C04413=1022.821,256.392,372.771,169.768,48.763,159.342
C04414=1022.827,256.640,372.742,169.772,48.759,159.342
C04415=1022.834,256.887,372.714,169.776,48.756,159.342
C04416=1022.841,257.136,372.685,169.779,48.751,159.342
C04417=1022.847,257.384,372.656,169.783,48.748,159.342
C04418=1022.853,257.632,372.627,169.787,48.744,159.341
C04419=1022.861,257.881,372.599,169.792,48.741,159.341
C04420=1022.867,258.129,372.570,169.796,48.737,159.341
C04421=1022.873,258.377,372.541,169.800,48.734,159.341
C04422=1022.880,258.625,372.512,169.804,48.730,159.341
C04423=1022.886,258.873,372.483,169.808,48.727,159.341
C04424=1022.892,259.121,372.454,169.812,48.723,159.340
C04425=1022.899,259.370,372.425,169.816,48.720,159.340
C04426=1022.906,259.618,372.396,169.820,48.716,159.340
C04427=1022.913,259.866,372.367,169.825,48.712,159.340
C04428=1022.919,260.114,372.338,169.829,48.709,159.340
C04429=1022.926,260.362,372.310,169.833,48.706,159.340
C04430=1022.933,260.611,372.280,169.838,48.702,159.339
C04431=1022.938,260.859,372.251,169.842,48.699,159.339
C04432=1022.944,261.107,372.222,169.846,48.696,159.339
C04433=1022.951,261.356,372.193,169.850,48.692,159.339
C04434=1022.957,261.604,372.164,169.854,48.689,159.339
C04435=1022.964,261.852,372.133,169.858,48.686,159.339
C04436=1022.970,262.100,372.104,169.862,48.682,159.339
C04437=1022.977,262.348,372.075,169.866,48.679,159.339
C04438=1022.983,262.596,372.046,169.870,48.676,159.338
C04439=1022.993,263.014,371.996,169.878,48.670,159.338
C04440=1023.005,263.433,371.947,169.884,48.664,159.338
C04441=1023.015,263.851,371.897,169.892,48.659,159.338
C04442=1023.025,264.269,371.847,169.899,48.653,159.338
C04443=1023.032,264.517,371.818,169.904,48.650,159.338
C04444=1023.039,264.765,371.788,169.908,48.647,159.338
C04445=1023.045,265.013,371.759,169.912,48.643,159.337
C04446=1023.051,265.262,371.730,169.916,48.641,159.337
C04447=1023.059,265.510,371.700,169.920,48.637,159.337
C04448=1023.065,265.758,371.671,169.925,48.634,159.337
C04449=1023.071,266.006,371.640,169.929,48.631,159.337
C04450=1023.077,266.255,371.611,169.933,48.627,159.337
C04451=1023.084,266.503,371.582,169.937,48.624,159.337
C04452=1023.090,266.750,371.552,169.941,48.621,159.337
C04453=1023.096,266.999,371.522,169.946,48.618,159.337
C04454=1023.103,267.247,371.492,169.950,48.615,159.337
C04455=1023.109,267.495,371.463,169.954,48.612,159.337
C04456=1023.116,267.744,371.433,169.958,48.608,159.336
C04457=1023.122,267.991,371.403,169.962,48.606,159.336
C04458=1023.128,268.239,371.374,169.967,48.602,159.336
C04459=1023.135,268.488,371.343,169.972,48.599,159.336
C04460=1023.141,268.736,371.314,169.976,48.596,159.336
C04461=1023.148,268.984,371.284,169.980,48.593,159.336
C04462=1023.155,269.232,371.254,169.984,48.590,159.336
C04463=1023.160,269.480,371.225,169.988,48.586,159.336
C04464=1023.167,269.728,371.195,169.993,48.584,159.336
C04465=1023.174,269.976,371.165,169.997,48.581,159.336
C04466=1023.180,270.225,371.135,170.001,48.577,159.336
C04467=1023.187,270.472,371.105,170.006,48.575,159.336
C04468=1023.193,270.721,371.074,170.010,48.572,159.336
C04469=1023.200,270.968,371.045,170.014,48.568,159.336
C04470=1023.205,271.217,371.015,170.018,48.566,159.336
C04471=1023.212,271.465,370.985,170.023,48.563,159.336
C04472=1023.218,271.713,370.954,170.027,48.560,159.336
C04473=1023.225,271.961,370.924,170.032,48.556,159.336
C04474=1023.231,272.209,370.894,170.036,48.553,159.336
C04475=1023.238,272.457,370.864,170.041,48.550,159.336
C04476=1023.244,272.706,370.834,170.045,48.548,159.336
C04477=1023.251,272.954,370.804,170.049,48.544,159.335
C04478=1023.257,273.202,370.774,170.054,48.541,159.335
C04479=1023.264,273.450,370.744,170.058,48.539,159.335
C04480=1023.270,273.698,370.713,170.062,48.536,159.335
C04481=1023.277,273.946,370.683,170.067,48.533,159.335
C04482=1023.283,274.194,370.653,170.071,48.530,159.335
C04483=1023.290,274.442,370.623,170.075,48.527,159.335
C04484=1023.296,274.690,370.592,170.079,48.524,159.335
C04485=1023.303,274.938,370.562,170.084,48.521,159.335
C04486=1023.309,275.186,370.532,170.089,48.518,159.335
C04487=1023.315,275.434,370.501,170.094,48.515,159.335
C04488=1023.322,275.682,370.471,170.098,48.512,159.335
C04489=1023.328,275.930,370.441,170.102,48.510,159.335
C04490=1023.335,276.178,370.411,170.107,48.507,159.335
C04491=1023.341,276.426,370.380,170.111,48.504,159.335
C04492=1023.348,276.675,370.350,170.115,48.501,159.335
C04493=1023.354,276.922,370.319,170.120,48.498,159.335
C04494=1023.361,277.170,370.288,170.124,48.496,159.335
C04495=1023.366,277.382,370.263,170.129,48.493,159.335
C04496=1023.372,277.593,370.237,170.132,48.490,159.335
C04497=1023.378,277.804,370.210,170.136,48.488,159.335
C04498=1023.382,278.016,370.184,170.139,48.486,159.335
C04499=1023.388,278.227,370.158,170.144,48.484,159.335
C04500=1023.394,278.439,370.132,170.147,48.481,159.335
C04501=1023.399,278.650,370.106,170.150,48.479,159.335
C04502=1023.405,278.861,370.080,170.155,48.477,159.336
C04503=1023.411,279.109,370.049,170.159,48.474,159.336
C04504=1023.418,279.358,370.018,170.164,48.471,159.336
C04505=1023.424,279.605,369.987,170.168,48.468,159.336
C04506=1023.430,279.853,369.957,170.173,48.465,159.336
C04507=1023.437,280.101,369.925,170.177,48.463,159.336
C04508=1023.444,280.349,369.895,170.182,48.460,159.336
C04509=1023.450,280.597,369.865,170.186,48.458,159.336
C04510=1023.457,280.845,369.833,170.190,48.455,159.336
C04511=1023.463,281.093,369.803,170.195,48.452,159.336
C04512=1023.469,281.341,369.772,170.200,48.450,159.336
C04513=1023.476,281.589,369.741,170.205,48.447,159.336
C04514=1023.483,281.837,369.710,170.209,48.444,159.336
C04515=1023.489,282.085,369.680,170.214,48.441,159.336
C04516=1023.496,282.333,369.648,170.218,48.439,159.336
C04517=1023.502,282.581,369.618,170.223,48.436,159.336
C04518=1023.509,282.829,369.586,170.227,48.433,159.336
C04519=1023.515,283.077,369.556,170.231,48.431,159.336
C04520=1023.522,283.325,369.525,170.236,48.428,159.336
C04521=1023.529,283.573,369.494,170.240,48.426,159.336
C04522=1023.535,283.821,369.463,170.246,48.423,159.336
C04523=1023.541,284.069,369.432,170.251,48.420,159.337
C04524=1023.548,284.317,369.401,170.255,48.418,159.337
C04525=1023.555,284.564,369.370,170.259,48.415,159.337
C04526=1023.562,284.813,369.339,170.264,48.413,159.337
C04527=1023.568,285.061,369.308,170.268,48.410,159.337
C04528=1023.575,285.309,369.277,170.273,48.408,159.337
C04529=1023.581,285.557,369.246,170.277,48.405,159.337
C04530=1023.588,285.804,369.215,170.283,48.403,159.337
C04531=1023.594,286.052,369.183,170.288,48.400,159.337
C04532=1023.601,286.300,369.152,170.292,48.398,159.337
C04533=1023.608,286.549,369.121,170.297,48.395,159.337
C04534=1023.614,286.797,369.090,170.301,48.393,159.338
C04535=1023.621,287.045,369.058,170.306,48.390,159.338
C04536=1023.627,287.292,369.027,170.310,48.388,159.338
C04537=1023.634,287.540,368.996,170.315,48.385,159.338
C04538=1023.641,287.788,368.964,170.319,48.383,159.338
C04539=1023.647,288.035,368.933,170.325,48.380,159.338
C04540=1023.654,288.283,368.902,170.330,48.378,159.338
C04541=1023.660,288.532,368.869,170.334,48.375,159.338
C04542=1023.667,288.779,368.838,170.339,48.373,159.338
C04543=1023.673,289.027,368.807,170.343,48.370,159.339
C04544=1023.680,289.275,368.775,170.348,48.368,159.339
C04545=1023.687,289.523,368.744,170.352,48.366,159.339
C04546=1023.694,289.771,368.712,170.357,48.363,159.339
C04547=1023.700,290.019,368.681,170.363,48.361,159.339
C04548=1023.706,290.267,368.649,170.367,48.358,159.339
C04549=1023.712,290.514,368.618,170.372,48.356,159.339
C04550=1023.719,290.762,368.586,170.377,48.354,159.340
C04551=1023.726,291.010,368.555,170.381,48.352,159.340
C04552=1023.733,291.258,368.523,170.386,48.349,159.340
C04553=1023.739,291.506,368.492,170.390,48.347,159.340
C04554=1023.746,291.754,368.461,170.396,48.344,159.340
C04555=1023.752,291.971,368.432,170.400,48.342,159.340
C04556=1023.758,292.189,368.404,170.404,48.340,159.341
C04557=1023.764,292.407,368.377,170.408,48.339,159.341
C04558=1023.769,292.624,368.349,170.413,48.336,159.341
C04559=1023.775,292.841,368.320,170.417,48.335,159.341
C04560=1023.781,293.059,368.293,170.421,48.332,159.341
C04561=1023.787,293.277,368.265,170.425,48.331,159.341
C04562=1023.793,293.493,368.237,170.430,48.328,159.341
C04563=1023.799,293.741,368.205,170.434,48.326,159.342
C04564=1023.805,293.989,368.173,170.439,48.324,159.342
C04565=1023.812,294.237,368.141,170.444,48.322,159.342
C04566=1023.818,294.485,368.109,170.448,48.320,159.342
C04567=1023.825,294.733,368.076,170.453,48.318,159.342
C04568=1023.832,294.981,368.045,170.458,48.316,159.343
C04569=1023.838,295.229,368.012,170.463,48.313,159.343
C04570=1023.844,295.477,367.980,170.468,48.311,159.343
C04571=1023.851,295.724,367.948,170.473,48.309,159.343
C04572=1023.858,295.972,367.915,170.478,48.307,159.343
C04573=1023.864,296.220,367.883,170.483,48.305,159.344
C04574=1023.871,296.467,367.851,170.487,48.303,159.344
C04575=1023.877,296.716,367.819,170.492,48.301,159.344
C04576=1023.884,296.963,367.787,170.497,48.299,159.344
C04577=1023.890,297.210,367.754,170.502,48.297,159.344
C04578=1023.897,297.459,367.722,170.507,48.294,159.345
C04579=1023.903,297.707,367.689,170.512,48.293,159.345
C04580=1023.910,297.954,367.657,170.517,48.291,159.345
C04581=1023.916,298.202,367.625,170.522,48.288,159.345
C04582=1023.923,298.450,367.592,170.526,48.286,159.346
C04583=1023.929,298.697,367.560,170.531,48.284,159.346
C04584=1023.937,298.945,367.527,170.536,48.283,159.346
C04585=1023.943,299.194,367.495,170.542,48.280,159.346
C04586=1023.950,299.441,367.463,170.547,48.278,159.347
C04587=1023.956,299.688,367.430,170.552,48.277,159.347
C04588=1023.962,299.936,367.397,170.556,48.274,159.347
C04589=1023.970,300.184,367.365,170.561,48.272,159.347
C04590=1023.976,300.432,367.333,170.566,48.270,159.348
C04591=1023.982,300.680,367.300,170.572,48.268,159.348
C04592=1023.989,300.927,367.268,170.577,48.266,159.348
C04593=1023.996,301.175,367.235,170.581,48.264,159.348
C04594=1024.003,301.423,367.203,170.586,48.263,159.349
C04595=1024.009,301.670,367.170,170.591,48.260,159.349
C04596=1024.016,301.919,367.137,170.597,48.259,159.349
C04597=1024.023,302.166,367.105,170.602,48.257,159.350
C04598=1024.030,302.413,367.072,170.606,48.254,159.350
C04599=1024.037,302.662,367.039,170.611,48.253,159.350
C04600=1024.044,302.909,367.007,170.616,48.251,159.350
C04601=1024.050,303.157,366.974,170.622,48.249,159.351
C04602=1024.057,303.405,366.941,170.627,48.247,159.351
C04603=1024.064,303.652,366.909,170.632,48.245,159.351
C04604=1024.070,303.900,366.876,170.637,48.243,159.351
C04605=1024.078,304.148,366.844,170.643,48.241,159.352
C04606=1024.084,304.395,366.811,170.647,48.239,159.352
C04607=1024.091,304.644,366.778,170.652,48.238,159.352
C04608=1024.098,304.891,366.746,170.657,48.236,159.353
C04609=1024.105,305.139,366.712,170.663,48.234,159.353
C04610=1024.111,305.386,366.679,170.668,48.232,159.353
C04611=1024.118,305.633,366.647,170.673,48.230,159.354
C04612=1024.125,305.882,366.614,170.678,48.228,159.354
C04613=1024.132,306.129,366.581,170.684,48.226,159.354
C04614=1024.139,306.377,366.548,170.689,48.225,159.355
C04615=1024.146,306.603,366.518,170.693,48.223,159.355
C04616=1024.152,306.829,366.489,170.697,48.221,159.355
C04617=1024.158,307.055,366.458,170.702,48.219,159.355
C04618=1024.164,307.281,366.427,170.707,48.218,159.356
C04619=1024.171,307.508,366.398,170.712,48.216,159.356
C04620=1024.177,307.733,366.368,170.717,48.215,159.356
C04621=1024.184,307.960,366.338,170.722,48.213,159.356
C04622=1024.190,308.186,366.307,170.726,48.211,159.357
C04623=1024.197,308.434,366.274,170.732,48.210,159.357
C04624=1024.204,308.681,366.242,170.737,48.208,159.357
C04625=1024.211,308.929,366.208,170.742,48.206,159.358
C04626=1024.218,309.178,366.175,170.748,48.204,159.358
C04627=1024.225,309.424,366.142,170.753,48.203,159.359
C04628=1024.232,309.672,366.109,170.758,48.201,159.359
C04629=1024.239,309.919,366.076,170.764,48.199,159.359
C04630=1024.246,310.167,366.043,170.769,48.197,159.359
C04631=1024.254,310.415,366.010,170.774,48.196,159.360
C04632=1024.260,310.663,365.977,170.779,48.194,159.360
C04633=1024.267,310.910,365.943,170.785,48.193,159.361
C04634=1024.273,311.158,365.909,170.790,48.191,159.361
C04635=1024.280,311.405,365.875,170.795,48.190,159.361
C04636=1024.286,311.653,365.842,170.800,48.188,159.362
C04637=1024.293,311.901,365.808,170.806,48.186,159.362
C04638=1024.300,312.149,365.774,170.811,48.185,159.363
C04639=1024.307,312.396,365.741,170.816,48.183,159.363
C04640=1024.314,312.643,365.707,170.821,48.182,159.363
C04641=1024.320,312.891,365.673,170.827,48.180,159.364
C04642=1024.327,313.139,365.640,170.832,48.179,159.364
C04643=1024.334,313.386,365.606,170.837,48.178,159.365
C04644=1024.340,313.633,365.572,170.843,48.176,159.365
C04645=1024.347,313.881,365.538,170.849,48.174,159.365
C04646=1024.354,314.129,365.504,170.854,48.173,159.366
C04647=1024.361,314.377,365.470,170.859,48.171,159.366
C04648=1024.367,314.624,365.436,170.864,48.171,159.367
C04649=1024.374,314.872,365.402,170.870,48.169,159.367
C04650=1024.382,315.119,365.369,170.875,48.167,159.367
C04651=1024.387,315.367,365.335,170.880,48.166,159.368
C04652=1024.395,315.614,365.301,170.886,48.165,159.368
C04653=1024.402,315.862,365.267,170.892,48.163,159.369
C04654=1024.409,316.109,365.232,170.897,48.162,159.369
C04655=1024.416,316.357,365.198,170.903,48.160,159.370
C04656=1024.422,316.604,365.164,170.908,48.159,159.370
C04657=1024.430,316.852,365.131,170.913,48.157,159.371
C04658=1024.436,317.100,365.096,170.919,48.156,159.371
C04659=1024.443,317.347,365.062,170.924,48.155,159.372
C04660=1024.450,317.595,365.029,170.929,48.153,159.372
C04661=1024.457,317.842,364.993,170.936,48.152,159.372
C04662=1024.464,318.089,364.960,170.941,48.151,159.373
C04663=1024.471,318.337,364.926,170.946,48.149,159.373
C04664=1024.478,318.585,364.892,170.952,48.148,159.374
C04665=1024.485,318.832,364.857,170.957,48.146,159.374
C04666=1024.492,319.080,364.823,170.963,48.146,159.375
C04667=1024.499,319.327,364.790,170.969,48.144,159.375
C04668=1024.506,319.575,364.754,170.974,48.143,159.376
C04669=1024.513,319.823,364.721,170.979,48.141,159.376
C04670=1024.521,320.070,364.687,170.985,48.140,159.377
C04671=1024.527,320.318,364.652,170.990,48.139,159.377
C04672=1024.535,320.565,364.618,170.997,48.138,159.378
C04673=1024.542,320.813,364.584,171.002,48.136,159.378
C04674=1024.549,321.060,364.549,171.007,48.135,159.379
C04675=1024.555,321.289,364.518,171.012,48.134,159.379
C04676=1024.562,321.518,364.486,171.018,48.133,159.380
C04677=1024.569,321.747,364.455,171.023,48.131,159.380
C04678=1024.575,321.975,364.422,171.028,48.131,159.380
C04679=1024.582,322.204,364.390,171.033,48.130,159.381
C04680=1024.588,322.432,364.359,171.038,48.128,159.381
C04681=1024.595,322.660,364.327,171.044,48.127,159.382
C04682=1024.601,322.890,364.295,171.049,48.126,159.382
C04683=1024.609,323.137,364.260,171.055,48.125,159.383
C04684=1024.616,323.385,364.226,171.061,48.124,159.383
C04685=1024.623,323.632,364.191,171.067,48.122,159.384
C04686=1024.630,323.880,364.157,171.072,48.121,159.384
C04687=1024.638,324.127,364.122,171.078,48.120,159.385
C04688=1024.645,324.375,364.087,171.084,48.119,159.386
C04689=1024.652,324.622,364.053,171.090,48.117,159.386
C04690=1024.659,324.869,364.019,171.095,48.116,159.387
C04691=1024.666,325.117,363.984,171.101,48.115,159.387
C04692=1024.674,325.365,363.950,171.107,48.114,159.388
C04693=1024.681,325.612,363.915,171.113,48.113,159.388
C04694=1024.688,325.860,363.880,171.118,48.112,159.389
C04695=1024.696,326.107,363.845,171.124,48.111,159.389
C04696=1024.703,326.355,363.811,171.130,48.110,159.390
C04697=1024.710,326.602,363.776,171.135,48.109,159.390
C04698=1024.718,326.850,363.741,171.142,48.108,159.391
C04699=1024.725,327.097,363.706,171.147,48.107,159.392
C04700=1024.733,327.345,363.671,171.153,48.106,159.392
C04701=1024.739,327.592,363.636,171.159,48.105,159.393
C04702=1024.746,327.839,363.601,171.165,48.104,159.393
C04703=1024.753,328.087,363.566,171.171,48.103,159.394
C04704=1024.761,328.334,363.531,171.177,48.102,159.394
C04705=1024.768,328.582,363.496,171.182,48.101,159.395
C04706=1024.775,328.829,363.460,171.189,48.100,159.396
C04707=1024.782,329.077,363.425,171.194,48.099,159.396
C04708=1024.789,329.324,363.390,171.201,48.098,159.397
C04709=1024.797,329.571,363.355,171.206,48.097,159.398
C04710=1024.804,329.819,363.319,171.212,48.096,159.398
C04711=1024.811,330.066,363.284,171.218,48.095,159.399
C04712=1024.818,330.313,363.248,171.224,48.094,159.399
C04713=1024.825,330.561,363.213,171.230,48.094,159.400
C04714=1024.833,330.808,363.178,171.236,48.093,159.401
C04715=1024.840,331.055,363.143,171.242,48.092,159.401
C04716=1024.847,331.303,363.107,171.248,48.091,159.402
C04717=1024.854,331.551,363.072,171.254,48.090,159.403
C04718=1024.862,331.798,363.036,171.260,48.089,159.403
C04719=1024.869,332.045,363.001,171.265,48.088,159.404
C04720=1024.877,332.292,362.965,171.272,48.088,159.405
C04721=1024.884,332.540,362.930,171.277,48.087,159.405
C04722=1024.891,332.787,362.894,171.284,48.086,159.406
C04723=1024.898,333.035,362.859,171.291,48.085,159.406
C04724=1024.906,333.282,362.824,171.296,48.084,159.407
C04725=1024.913,333.529,362.788,171.303,48.084,159.408
C04726=1024.921,333.777,362.752,171.308,48.083,159.408
C04727=1024.928,334.024,362.716,171.315,48.082,159.409
C04728=1024.935,334.271,362.680,171.320,48.082,159.410
C04729=1024.942,334.518,362.644,171.327,48.081,159.411
C04730=1024.950,334.766,362.609,171.332,48.080,159.411
C04731=1024.957,335.013,362.573,171.339,48.080,159.412
C04732=1024.964,335.261,362.536,171.345,48.079,159.413
C04733=1024.971,335.507,362.500,171.351,48.078,159.413
C04734=1024.978,335.756,362.465,171.358,48.078,159.414
C04735=1024.985,335.981,362.432,171.363,48.077,159.415
C04736=1024.992,336.209,362.399,171.369,48.077,159.415
C04737=1024.999,336.435,362.366,171.374,48.076,159.416
C04738=1025.005,336.661,362.334,171.380,48.075,159.417
C04739=1025.012,336.887,362.300,171.385,48.075,159.417
C04740=1025.020,337.114,362.267,171.392,48.074,159.418
C04741=1025.025,337.341,362.234,171.397,48.074,159.419
C04742=1025.032,337.567,362.201,171.403,48.073,159.419
C04743=1025.040,337.814,362.165,171.408,48.073,159.420
C04744=1025.047,338.061,362.128,171.415,48.072,159.421
C04745=1025.055,338.309,362.092,171.422,48.071,159.422
C04746=1025.062,338.556,362.056,171.427,48.071,159.422
C04747=1025.070,338.803,362.020,171.434,48.070,159.423
C04748=1025.077,339.050,361.984,171.441,48.070,159.424
C04749=1025.085,339.298,361.948,171.446,48.069,159.424
C04750=1025.092,339.545,361.912,171.453,48.069,159.425
C04751=1025.100,339.792,361.876,171.460,48.068,159.426
C04752=1025.107,340.040,361.839,171.465,48.068,159.427
C04753=1025.115,340.287,361.802,171.472,48.067,159.428
C04754=1025.122,340.533,361.766,171.479,48.067,159.428
C04755=1025.130,340.781,361.730,171.484,48.067,159.429
C04756=1025.137,341.029,361.693,171.491,48.066,159.430
C04757=1025.145,341.275,361.656,171.498,48.065,159.431
C04758=1025.152,341.523,361.620,171.504,48.065,159.431
C04759=1025.159,341.771,361.583,171.510,48.065,159.432
C04760=1025.166,342.017,361.547,171.517,48.064,159.433
C04761=1025.174,342.264,361.510,171.523,48.064,159.434
C04762=1025.181,342.511,361.473,171.529,48.063,159.435
C04763=1025.189,342.759,361.437,171.536,48.063,159.436
C04764=1025.197,343.006,361.400,171.543,48.063,159.436
C04765=1025.204,343.253,361.363,171.549,48.063,159.437
C04766=1025.212,343.501,361.327,171.555,48.062,159.438
C04767=1025.220,343.748,361.290,171.562,48.062,159.439
C04768=1025.227,343.995,361.252,171.568,48.062,159.440
C04769=1025.235,344.242,361.216,171.575,48.061,159.440
C04770=1025.242,344.489,361.178,171.582,48.061,159.441
C04771=1025.250,344.737,361.142,171.589,48.061,159.442
C04772=1025.257,344.984,361.105,171.594,48.060,159.443
C04773=1025.265,345.231,361.068,171.601,48.060,159.444
C04774=1025.272,345.478,361.032,171.608,48.060,159.445
C04775=1025.280,345.725,360.994,171.615,48.059,159.446
C04776=1025.288,345.972,360.957,171.622,48.059,159.447
C04777=1025.295,346.219,360.920,171.627,48.059,159.447
C04778=1025.303,346.467,360.883,171.634,48.059,159.448
C04779=1025.311,346.714,360.846,171.641,48.059,159.449
C04780=1025.318,346.961,360.809,171.648,48.058,159.450
C04781=1025.326,347.208,360.772,171.654,48.058,159.451
C04782=1025.333,347.455,360.734,171.661,48.058,159.452
C04783=1025.341,347.702,360.697,171.668,48.058,159.453
C04784=1025.349,347.949,360.660,171.675,48.058,159.454
C04785=1025.357,348.196,360.623,171.681,48.057,159.454
C04786=1025.364,348.443,360.585,171.688,48.058,159.455
C04787=1025.372,348.690,360.548,171.694,48.058,159.456
C04788=1025.379,348.937,360.511,171.701,48.057,159.457
C04789=1025.387,349.184,360.473,171.708,48.057,159.458
C04790=1025.395,349.432,360.436,171.715,48.057,159.459
C04791=1025.402,349.679,360.398,171.722,48.057,159.460
C04792=1025.410,349.926,360.361,171.729,48.057,159.461
C04793=1025.418,350.172,360.323,171.735,48.057,159.462
C04794=1025.425,350.420,360.286,171.742,48.057,159.463
C04795=1025.432,350.645,360.252,171.749,48.057,159.464
C04796=1025.439,350.870,360.217,171.755,48.057,159.465
C04797=1025.446,351.094,360.182,171.761,48.057,159.465
C04798=1025.453,351.320,360.148,171.767,48.057,159.466
C04799=1025.461,351.544,360.114,171.773,48.057,159.467
C04800=1025.468,351.770,360.080,171.779,48.057,159.468
C04801=1025.475,351.994,360.046,171.786,48.057,159.469
C04802=1025.481,352.219,360.011,171.792,48.057,159.470
C04803=1025.490,352.466,359.973,171.799,48.057,159.471
C04804=1025.497,352.713,359.935,171.806,48.057,159.472
C04805=1025.505,352.960,359.898,171.813,48.057,159.473
C04806=1025.514,353.207,359.860,171.820,48.058,159.474
C04807=1025.521,353.454,359.822,171.827,48.058,159.475
C04808=1025.529,353.701,359.784,171.834,48.058,159.476
C04809=1025.536,353.948,359.746,171.841,48.058,159.477
C04810=1025.545,354.195,359.708,171.848,48.058,159.478
C04811=1025.552,354.442,359.670,171.855,48.058,159.479
C04812=1025.560,354.689,359.632,171.862,48.058,159.480
C04813=1025.568,354.936,359.594,171.869,48.058,159.481
C04814=1025.576,355.183,359.557,171.877,48.058,159.482
C04815=1025.584,355.430,359.518,171.884,48.059,159.483
C04816=1025.592,355.677,359.480,171.891,48.059,159.484
C04817=1025.600,355.924,359.441,171.898,48.059,159.485
C04818=1025.607,356.170,359.403,171.905,48.059,159.486
C04819=1025.615,356.418,359.365,171.912,48.059,159.487
C04820=1025.623,356.665,359.327,171.919,48.059,159.488
C04821=1025.631,356.912,359.288,171.927,48.060,159.489
C04822=1025.639,357.159,359.250,171.934,48.060,159.490
C04823=1025.647,357.405,359.212,171.941,48.061,159.491
C04824=1025.656,357.653,359.173,171.948,48.061,159.492
C04825=1025.663,357.899,359.135,171.955,48.061,159.493
C04826=1025.671,358.146,359.097,171.962,48.061,159.495
C04827=1025.679,358.393,359.058,171.969,48.061,159.496
C04828=1025.687,358.640,359.020,171.977,48.062,159.497
C04829=1025.695,358.887,358.981,171.984,48.062,159.498
C04830=1025.704,359.134,358.942,171.991,48.063,159.499
C04831=1025.711,359.380,358.903,171.998,48.063,159.500
C04832=1025.719,359.628,358.865,172.005,48.063,159.501
C04833=1025.727,359.875,358.826,172.013,48.064,159.502
C04834=1025.735,360.121,358.788,172.021,48.064,159.503
C04835=1025.743,360.368,358.749,172.028,48.064,159.505
C04836=1025.752,360.615,358.710,172.036,48.065,159.506
C04837=1025.760,360.862,358.671,172.043,48.066,159.507
C04838=1025.768,361.108,358.633,172.050,48.066,159.508
C04839=1025.775,361.356,358.593,172.057,48.066,159.509
C04840=1025.784,361.602,358.554,172.065,48.067,159.510
C04841=1025.792,361.849,358.515,172.072,48.068,159.512
C04842=1025.800,362.096,358.476,172.079,48.068,159.513
C04843=1025.807,362.342,358.436,172.088,48.069,159.514
C04844=1025.815,362.590,358.398,172.095,48.069,159.515
C04845=1025.824,362.836,358.359,172.103,48.070,159.516
C04846=1025.832,363.083,358.320,172.110,48.070,159.518
C04847=1025.840,363.330,358.281,172.117,48.071,159.519
C04848=1025.848,363.577,358.241,172.126,48.071,159.520
C04849=1025.856,363.823,358.202,172.133,48.072,159.521
C04850=1025.864,364.070,358.163,172.140,48.073,159.522
C04851=1025.873,364.317,358.124,172.148,48.073,159.524
C04852=1025.880,364.563,358.084,172.155,48.074,159.525
C04853=1025.889,364.810,358.045,172.163,48.074,159.526
C04854=1025.897,365.057,358.006,172.171,48.075,159.527
C04855=1025.905,365.285,357.969,172.178,48.076,159.528
C04856=1025.913,365.513,357.933,172.184,48.076,159.530
C04857=1025.920,365.742,357.897,172.192,48.077,159.531
C04858=1025.928,365.970,357.860,172.199,48.078,159.532
C04859=1025.935,366.198,357.823,172.206,48.078,159.533
C04860=1025.943,366.427,357.786,172.214,48.078,159.534
C04861=1025.951,366.655,357.750,172.220,48.079,159.535
C04862=1025.959,366.884,357.714,172.227,48.080,159.536
C04863=1025.967,367.130,357.674,172.236,48.081,159.538
C04864=1025.976,367.376,357.634,172.243,48.081,159.539
C04865=1025.984,367.623,357.594,172.251,48.082,159.540
C04866=1025.992,367.870,357.555,172.259,48.083,159.542
C04867=1026.000,368.116,357.516,172.267,48.084,159.543
C04868=1026.009,368.363,357.476,172.274,48.085,159.544
C04869=1026.017,368.610,357.436,172.283,48.085,159.545
C04870=1026.026,368.856,357.396,172.291,48.086,159.547
C04871=1026.034,369.103,357.356,172.298,48.087,159.548
C04872=1026.042,369.350,357.317,172.307,48.088,159.549
C04873=1026.050,369.596,357.276,172.314,48.088,159.551
C04874=1026.059,369.843,357.237,172.323,48.089,159.552
C04875=1026.067,370.090,357.196,172.330,48.091,159.554
C04876=1026.076,370.336,357.157,172.338,48.091,159.555
C04877=1026.084,370.583,357.116,172.346,48.092,159.556
C04878=1026.092,370.829,357.075,172.354,48.093,159.558
C04879=1026.101,371.076,357.036,172.363,48.094,159.559
C04880=1026.109,371.323,356.995,172.370,48.095,159.560
C04881=1026.117,371.569,356.956,172.378,48.096,159.562
C04882=1026.126,371.816,356.915,172.387,48.097,159.563
C04883=1026.135,372.062,356.875,172.394,48.098,159.564
C04884=1026.143,372.308,356.834,172.403,48.099,159.566
C04885=1026.151,372.556,356.794,172.411,48.100,159.567
C04886=1026.160,372.802,356.754,172.419,48.101,159.569
C04887=1026.168,373.049,356.713,172.427,48.102,159.570
C04888=1026.177,373.295,356.673,172.436,48.103,159.572
C04889=1026.185,373.541,356.632,172.443,48.104,159.573
C04890=1026.194,373.788,356.591,172.452,48.105,159.574
C04891=1026.203,374.034,356.551,172.460,48.107,159.576
C04892=1026.211,374.282,356.511,172.469,48.107,159.577
C04893=1026.220,374.528,356.471,172.476,48.109,159.579
C04894=1026.228,374.775,356.430,172.485,48.109,159.580
C04895=1026.237,375.020,356.389,172.494,48.110,159.581
C04896=1026.246,375.267,356.348,172.501,48.112,159.583
C04897=1026.255,375.514,356.307,172.510,48.113,159.585
C04898=1026.263,375.760,356.267,172.518,48.114,159.586
C04899=1026.272,376.007,356.226,172.527,48.115,159.587
C04900=1026.281,376.253,356.186,172.535,48.116,159.589
C04901=1026.289,376.500,356.145,172.544,48.118,159.590
C04902=1026.298,376.746,356.103,172.552,48.119,159.592
C04903=1026.307,376.992,356.063,172.560,48.120,159.593
C04904=1026.316,377.239,356.022,172.569,48.121,159.595
C04905=1026.325,377.486,355.980,172.578,48.122,159.596
C04906=1026.333,377.732,355.940,172.586,48.124,159.598
C04907=1026.342,377.978,355.898,172.594,48.125,159.599
C04908=1026.350,378.225,355.857,172.603,48.126,159.601
C04909=1026.359,378.471,355.816,172.611,48.128,159.603
C04910=1026.367,378.718,355.775,172.620,48.129,159.604
C04911=1026.376,378.964,355.733,172.629,48.131,159.606
C04912=1026.385,379.210,355.692,172.637,48.132,159.607
C04913=1026.394,379.457,355.651,172.646,48.133,159.609
C04914=1026.403,379.703,355.609,172.655,48.135,159.610
C04915=1026.412,379.942,355.569,172.663,48.136,159.612
C04916=1026.420,380.181,355.529,172.672,48.137,159.613
C04917=1026.429,380.420,355.488,172.681,48.139,159.615
C04918=1026.437,380.658,355.449,172.688,48.140,159.616
C04919=1026.446,380.897,355.408,172.698,48.141,159.618
C04920=1026.453,381.136,355.368,172.706,48.143,159.620
C04921=1026.462,381.375,355.327,172.714,48.144,159.621
C04922=1026.471,381.614,355.287,172.722,48.146,159.623
C04923=1026.480,381.860,355.245,172.731,48.147,159.624
C04924=1026.489,382.106,355.204,172.740,48.149,159.626
C04925=1026.498,382.352,355.162,172.749,48.150,159.628
C04926=1026.507,382.599,355.120,172.758,48.152,159.629
C04927=1026.516,382.845,355.079,172.768,48.153,159.631
C04928=1026.525,383.092,355.037,172.777,48.154,159.633
C04929=1026.534,383.338,354.995,172.785,48.156,159.634
C04930=1026.543,383.584,354.953,172.794,48.158,159.636
C04931=1026.552,383.831,354.912,172.803,48.160,159.638
C04932=1026.561,384.076,354.869,172.812,48.161,159.639
C04933=1026.571,384.323,354.827,172.821,48.163,159.641
C04934=1026.580,384.570,354.786,172.830,48.164,159.643
C04935=1026.589,384.816,354.743,172.840,48.166,159.645
C04936=1026.598,385.062,354.701,172.849,48.168,159.646
C04937=1026.607,385.308,354.660,172.858,48.169,159.648
C04938=1026.616,385.554,354.617,172.867,48.171,159.650
C04939=1026.626,385.801,354.575,172.876,48.172,159.651
C04940=1026.635,386.047,354.533,172.885,48.174,159.653
C04941=1026.644,386.293,354.491,172.894,48.176,159.655
C04942=1026.653,386.539,354.449,172.904,48.178,159.657
C04943=1026.663,386.786,354.406,172.913,48.179,159.658
C04944=1026.672,387.032,354.364,172.922,48.181,159.660
C04945=1026.681,387.277,354.322,172.931,48.183,159.662
C04946=1026.689,387.524,354.279,172.941,48.185,159.664
C04947=1026.699,387.771,354.237,172.950,48.187,159.666
C04948=1026.708,388.016,354.194,172.960,48.189,159.668
C04949=1026.718,388.262,354.152,172.970,48.190,159.669
C04950=1026.727,388.509,354.109,172.979,48.192,159.671
C04951=1026.736,388.755,354.066,172.988,48.194,159.673
C04952=1026.746,389.001,354.023,172.998,48.196,159.675
C04953=1026.755,389.247,353.981,173.007,48.198,159.677
C04954=1026.764,389.492,353.938,173.016,48.199,159.678
C04955=1026.773,389.739,353.895,173.026,48.201,159.680
C04956=1026.783,389.985,353.852,173.036,48.203,159.682
C04957=1026.792,390.231,353.810,173.045,48.205,159.684
C04958=1026.801,390.477,353.766,173.055,48.208,159.686
C04959=1026.811,390.723,353.723,173.064,48.210,159.688
C04960=1026.820,390.969,353.681,173.074,48.212,159.690
C04961=1026.830,391.215,353.636,173.084,48.213,159.692
C04962=1026.839,391.461,353.594,173.094,48.215,159.694
C04963=1026.848,391.708,353.551,173.103,48.217,159.695
C04964=1026.858,391.954,353.507,173.113,48.220,159.697
C04965=1026.867,392.199,353.465,173.123,48.222,159.699
C04966=1026.877,392.445,353.421,173.133,48.224,159.701
C04967=1026.886,392.691,353.378,173.142,48.226,159.703
C04968=1026.896,392.937,353.335,173.153,48.228,159.705
C04969=1026.905,393.184,353.291,173.162,48.230,159.707
C04970=1026.915,393.430,353.248,173.172,48.232,159.709
C04971=1026.924,393.675,353.204,173.182,48.234,159.711
C04972=1026.934,393.921,353.161,173.192,48.237,159.713
C04973=1026.943,394.168,353.117,173.201,48.239,159.715
C04974=1026.953,394.413,353.074,173.212,48.241,159.717
C04975=1026.964,394.681,353.026,173.223,48.243,159.719
C04976=1026.973,394.949,352.978,173.234,48.246,159.722
C04977=1026.984,395.216,352.931,173.245,48.248,159.724
C04978=1026.995,395.484,352.883,173.255,48.250,159.726
C04979=1027.004,395.731,352.839,173.266,48.253,159.728
C04980=1027.015,395.976,352.795,173.276,48.255,159.730
C04981=1027.023,396.222,352.752,173.286,48.258,159.732
C04982=1027.033,396.468,352.708,173.296,48.260,159.734
C04983=1027.043,396.714,352.664,173.307,48.262,159.736
C04984=1027.053,396.960,352.620,173.316,48.264,159.738
C04985=1027.063,397.205,352.576,173.327,48.266,159.740
C04986=1027.073,397.451,352.532,173.337,48.269,159.742
C04987=1027.082,397.697,352.488,173.348,48.272,159.745
C04988=1027.092,397.943,352.444,173.358,48.274,159.747
C04989=1027.102,398.188,352.400,173.369,48.277,159.749
C04990=1027.112,398.435,352.356,173.379,48.279,159.751
C04991=1027.122,398.680,352.311,173.389,48.281,159.753
C04992=1027.132,398.927,352.267,173.400,48.283,159.755
C04993=1027.142,399.172,352.222,173.410,48.287,159.758
C04994=1027.151,399.418,352.178,173.421,48.289,159.760
C04995=1027.162,399.663,352.134,173.431,48.291,159.762
C04996=1027.171,399.910,352.090,173.441,48.294,159.764
C04997=1027.181,400.155,352.045,173.452,48.296,159.766
C04998=1027.191,400.401,352.000,173.463,48.299,159.769
C04999=1027.202,400.647,351.955,173.474,48.301,159.771
C05000=1027.211,400.892,351.911,173.484,48.304,159.773
C05001=1027.221,401.138,351.866,173.495,48.307,159.775
C05002=1027.230,401.384,351.822,173.506,48.309,159.777
C05003=1027.241,401.630,351.776,173.517,48.312,159.780
C05004=1027.251,401.875,351.732,173.527,48.315,159.782
C05005=1027.261,402.121,351.687,173.538,48.317,159.784
C05006=1027.271,402.367,351.642,173.549,48.320,159.787
C05007=1027.281,402.612,351.597,173.560,48.322,159.789
C05008=1027.291,402.857,351.552,173.571,48.325,159.791
C05009=1027.301,403.103,351.507,173.582,48.328,159.793
C05010=1027.311,403.349,351.462,173.592,48.331,159.796
C05011=1027.322,403.595,351.416,173.603,48.334,159.798
C05012=1027.331,403.840,351.371,173.614,48.336,159.800
C05013=1027.342,404.086,351.326,173.625,48.339,159.803
C05014=1027.352,404.331,351.280,173.636,48.342,159.805
C05015=1027.362,404.577,351.235,173.647,48.345,159.807
C05016=1027.372,404.822,351.190,173.659,48.348,159.810
C05017=1027.382,405.068,351.144,173.670,48.351,159.812
C05018=1027.393,405.314,351.098,173.681,48.353,159.815
C05019=1027.403,405.560,351.054,173.692,48.356,159.817
C05020=1027.413,405.805,351.008,173.704,48.360,159.820
C05021=1027.423,406.050,350.962,173.715,48.362,159.822
C05022=1027.434,406.296,350.917,173.726,48.365,159.824
C05023=1027.444,406.542,350.871,173.737,48.368,159.827
C05024=1027.455,406.787,350.825,173.748,48.371,159.829
C05025=1027.465,407.032,350.780,173.761,48.374,159.832
C05026=1027.475,407.279,350.734,173.772,48.377,159.834
C05027=1027.486,407.524,350.689,173.783,48.380,159.837
C05028=1027.496,407.770,350.643,173.795,48.383,159.839
C05029=1027.507,408.015,350.597,173.806,48.386,159.842
C05030=1027.518,408.261,350.551,173.818,48.389,159.844
C05031=1027.528,408.507,350.505,173.830,48.392,159.847
C05032=1027.539,408.752,350.459,173.841,48.395,159.849
C05033=1027.550,408.998,350.413,173.853,48.398,159.852
C05034=1027.560,409.243,350.367,173.865,48.401,159.854
C05035=1027.572,409.533,350.313,173.878,48.405,159.857
C05036=1027.585,409.822,350.259,173.892,48.409,159.860
C05037=1027.598,410.113,350.204,173.906,48.412,159.863
C05038=1027.610,410.402,350.148,173.920,48.416,159.866
C05039=1027.621,410.648,350.102,173.932,48.419,159.869
C05040=1027.632,410.893,350.056,173.944,48.422,159.872
C05041=1027.642,411.138,350.009,173.956,48.426,159.874
C05042=1027.653,411.383,349.963,173.968,48.429,159.877
C05043=1027.664,411.628,349.916,173.980,48.432,159.879
C05044=1027.674,411.875,349.869,173.992,48.436,159.882
C05045=1027.685,412.120,349.823,174.004,48.439,159.885
C05046=1027.696,412.365,349.776,174.016,48.443,159.888
C05047=1027.706,412.610,349.729,174.028,48.446,159.890
C05048=1027.717,412.857,349.682,174.040,48.450,159.893
C05049=1027.728,413.102,349.636,174.053,48.452,159.896
C05050=1027.738,413.347,349.589,174.066,48.456,159.898
C05051=1027.750,413.592,349.542,174.077,48.459,159.901
C05052=1027.761,413.837,349.495,174.090,48.463,159.904
C05053=1027.771,414.083,349.448,174.102,48.466,159.907
C05054=1027.783,414.328,349.401,174.114,48.470,159.910
C05055=1027.794,414.573,349.353,174.127,48.473,159.912
C05056=1027.805,414.818,349.306,174.139,48.477,159.915
C05057=1027.816,415.064,349.259,174.152,48.480,159.918
C05058=1027.827,415.309,349.212,174.164,48.483,159.921
C05059=1027.838,415.555,349.164,174.177,48.487,159.923
C05060=1027.849,415.800,349.117,174.189,48.491,159.926
C05061=1027.861,416.045,349.070,174.202,48.494,159.929
C05062=1027.872,416.291,349.022,174.215,48.498,159.932
C05063=1027.883,416.536,348.975,174.228,48.502,159.935
C05064=1027.894,416.781,348.927,174.241,48.505,159.938
C05065=1027.905,417.026,348.879,174.254,48.509,159.941
C05066=1027.916,417.271,348.832,174.266,48.513,159.944
C05067=1027.927,417.517,348.784,174.279,48.516,159.946
C05068=1027.939,417.762,348.736,174.292,48.520,159.949
C05069=1027.949,418.007,348.688,174.305,48.524,159.952
C05070=1027.961,418.252,348.641,174.318,48.528,159.955
C05071=1027.972,418.497,348.592,174.331,48.532,159.958
C05072=1027.983,418.742,348.544,174.344,48.535,159.961
C05073=1027.995,418.987,348.496,174.357,48.539,159.964
C05074=1028.006,419.233,348.448,174.370,48.543,159.967
C05075=1028.017,419.478,348.400,174.383,48.547,159.970
C05076=1028.029,419.722,348.352,174.396,48.550,159.973
C05077=1028.040,419.968,348.304,174.410,48.554,159.976
C05078=1028.052,420.213,348.256,174.424,48.558,159.979
C05079=1028.063,420.458,348.207,174.437,48.562,159.983
C05080=1028.075,420.703,348.159,174.450,48.566,159.986
C05081=1028.086,420.949,348.111,174.463,48.570,159.989
C05082=1028.098,421.193,348.062,174.478,48.574,159.992
C05083=1028.110,421.439,348.014,174.491,48.578,159.995
C05084=1028.121,421.683,347.965,174.504,48.582,159.998
C05085=1028.133,421.928,347.918,174.517,48.586,160.001
C05086=1028.144,422.173,347.869,174.532,48.590,160.005
C05087=1028.156,422.418,347.819,174.545,48.594,160.008
C05088=1028.167,422.664,347.771,174.560,48.598,160.011
C05089=1028.180,422.908,347.722,174.573,48.602,160.014
C05090=1028.191,423.153,347.673,174.586,48.606,160.017
C05091=1028.203,423.398,347.624,174.601,48.610,160.020
C05092=1028.214,423.643,347.575,174.614,48.614,160.024
C05093=1028.226,423.888,347.526,174.629,48.618,160.027
C05094=1028.239,424.133,347.477,174.642,48.623,160.030
C05095=1028.250,424.360,347.431,174.655,48.626,160.033
C05096=1028.260,424.588,347.386,174.668,48.630,160.036
C05097=1028.271,424.814,347.339,174.682,48.634,160.039
C05098=1028.283,425.042,347.295,174.695,48.638,160.043
C05099=1028.293,425.269,347.248,174.708,48.642,160.046
C05100=1028.304,425.496,347.202,174.722,48.646,160.049
C05101=1028.315,425.723,347.157,174.735,48.650,160.052
C05102=1028.327,425.950,347.111,174.748,48.654,160.055
C05103=1028.339,426.194,347.062,174.762,48.658,160.058
C05104=1028.351,426.439,347.012,174.777,48.663,160.062
C05105=1028.363,426.684,346.962,174.791,48.667,160.065
C05106=1028.375,426.928,346.912,174.806,48.672,160.069
C05107=1028.387,427.174,346.863,174.820,48.676,160.072
C05108=1028.399,427.418,346.813,174.835,48.681,160.075
C05109=1028.411,427.663,346.763,174.849,48.685,160.079
C05110=1028.423,427.907,346.713,174.864,48.689,160.082
C05111=1028.435,428.152,346.663,174.879,48.694,160.086
C05112=1028.448,428.397,346.613,174.894,48.698,160.089
C05113=1028.459,428.642,346.562,174.908,48.702,160.093
C05114=1028.471,428.886,346.512,174.923,48.707,160.096
C05115=1028.483,429.131,346.462,174.938,48.712,160.100
C05116=1028.496,429.375,346.412,174.953,48.716,160.103
C05117=1028.508,429.620,346.361,174.968,48.721,160.107
C05118=1028.520,429.865,346.311,174.983,48.725,160.111
C05119=1028.533,430.109,346.261,174.999,48.730,160.114
C05120=1028.545,430.354,346.210,175.014,48.735,160.118
C05121=1028.558,430.599,346.160,175.029,48.739,160.122
C05122=1028.570,430.843,346.110,175.044,48.744,160.125
C05123=1028.583,431.088,346.058,175.060,48.749,160.129
C05124=1028.596,431.333,346.008,175.076,48.753,160.133
C05125=1028.608,431.577,345.957,175.091,48.758,160.136
C05126=1028.621,431.821,345.907,175.106,48.763,160.140
C05127=1028.633,432.066,345.857,175.122,48.768,160.144
C05128=1028.647,432.311,345.805,175.137,48.773,160.148
C05129=1028.659,432.555,345.755,175.153,48.778,160.151
C05130=1028.672,432.799,345.704,175.169,48.782,160.155
C05131=1028.685,433.044,345.653,175.184,48.787,160.159
C05132=1028.697,433.289,345.601,175.200,48.792,160.163
C05133=1028.710,433.534,345.550,175.216,48.797,160.166
C05134=1028.723,433.778,345.499,175.232,48.801,160.170
C05135=1028.740,434.113,345.428,175.254,48.808,160.176
C05136=1028.759,434.447,345.358,175.276,48.815,160.181
C05137=1028.776,434.783,345.288,175.298,48.822,160.186
C05138=1028.794,435.118,345.217,175.321,48.828,160.192
C05139=1028.807,435.362,345.165,175.337,48.834,160.196
C05140=1028.820,435.607,345.114,175.353,48.839,160.200
C05141=1028.832,435.851,345.061,175.370,48.844,160.204
C05142=1028.846,436.095,345.009,175.386,48.849,160.208
C05143=1028.859,436.339,344.958,175.403,48.854,160.212
C05144=1028.872,436.584,344.905,175.420,48.860,160.216
C05145=1028.885,436.828,344.854,175.436,48.865,160.220
C05146=1028.899,437.072,344.802,175.453,48.870,160.224
C05147=1028.912,437.317,344.749,175.470,48.875,160.228
C05148=1028.924,437.560,344.698,175.486,48.880,160.232
C05149=1028.938,437.805,344.646,175.503,48.885,160.236
C05150=1028.951,438.049,344.593,175.520,48.891,160.240
C05151=1028.965,438.293,344.541,175.537,48.896,160.245
C05152=1028.978,438.537,344.489,175.554,48.901,160.249
C05153=1028.991,438.782,344.436,175.571,48.906,160.253
C05154=1029.005,439.025,344.384,175.588,48.912,160.257
C05155=1029.020,439.296,344.325,175.607,48.918,160.262
C05156=1029.035,439.567,344.267,175.627,48.924,160.267
C05157=1029.049,439.836,344.209,175.646,48.930,160.271
C05158=1029.065,440.107,344.150,175.665,48.936,160.276
C05159=1029.078,440.351,344.097,175.683,48.941,160.280
C05160=1029.092,440.594,344.044,175.700,48.947,160.285
C05161=1029.105,440.839,343.991,175.718,48.952,160.289
C05162=1029.119,441.082,343.938,175.735,48.958,160.293
C05163=1029.132,441.326,343.885,175.754,48.963,160.298
C05164=1029.147,441.571,343.832,175.771,48.969,160.302
C05165=1029.161,441.814,343.779,175.789,48.974,160.307
C05166=1029.174,442.058,343.726,175.807,48.980,160.311
C05167=1029.188,442.302,343.673,175.825,48.985,160.316
C05168=1029.202,442.546,343.619,175.843,48.991,160.320
C05169=1029.216,442.789,343.566,175.861,48.997,160.325
C05170=1029.230,443.033,343.512,175.879,49.002,160.329
C05171=1029.244,443.276,343.459,175.898,49.008,160.334
C05172=1029.259,443.519,343.407,175.916,49.013,160.338
C05173=1029.275,443.762,343.354,175.934,49.019,160.343
C05174=1029.291,444.006,343.303,175.952,49.024,160.347
C05175=1029.307,444.249,343.252,175.972,49.029,160.352
C05176=1029.323,444.493,343.201,175.990,49.035,160.356
C05177=1029.341,444.737,343.150,176.009,49.039,160.360
C05178=1029.359,444.981,343.100,176.028,49.045,160.365
C05179=1029.377,445.225,343.051,176.047,49.050,160.369
C05180=1029.395,445.469,343.001,176.066,49.055,160.374
C05181=1029.415,445.712,342.952,176.085,49.059,160.378
C05182=1029.435,445.957,342.904,176.104,49.064,160.383
C05183=1029.455,446.201,342.856,176.124,49.068,160.387
C05184=1029.476,446.445,342.808,176.143,49.073,160.392
C05185=1029.497,446.690,342.761,176.162,49.078,160.396
C05186=1029.518,446.934,342.714,176.182,49.082,160.400
C05187=1029.541,447.179,342.668,176.201,49.087,160.405
C05188=1029.563,447.423,342.621,176.221,49.091,160.409
C05189=1029.586,447.668,342.575,176.241,49.095,160.414
C05190=1029.609,447.913,342.530,176.261,49.099,160.418
C05191=1029.634,448.158,342.485,176.281,49.104,160.422
C05192=1029.658,448.403,342.442,176.301,49.108,160.427
C05193=1029.682,448.647,342.397,176.321,49.112,160.431
C05194=1029.708,448.893,342.354,176.341,49.115,160.435
C05195=1029.734,449.138,342.310,176.361,49.120,160.440
C05196=1029.761,449.383,342.268,176.382,49.123,160.444
C05197=1029.788,449.628,342.225,176.402,49.127,160.449
C05198=1029.815,449.873,342.183,176.422,49.131,160.453
C05199=1029.843,450.119,342.141,176.443,49.134,160.457
C05200=1029.871,450.364,342.101,176.464,49.138,160.462
C05201=1029.900,450.609,342.060,176.485,49.142,160.466
C05202=1029.929,450.854,342.020,176.505,49.145,160.470
C05203=1029.958,451.100,341.979,176.527,49.148,160.475
C05204=1029.990,451.345,341.939,176.548,49.151,160.479
C05205=1030.020,451.591,341.901,176.569,49.154,160.483
C05206=1030.051,451.837,341.862,176.590,49.158,160.488
C05207=1030.083,452.082,341.823,176.612,49.161,160.492
C05208=1030.115,452.328,341.786,176.633,49.164,160.496
C05209=1030.147,452.573,341.748,176.655,49.167,160.501
C05210=1030.181,452.818,341.711,176.677,49.169,160.505
C05211=1030.215,453.065,341.674,176.698,49.173,160.509
C05212=1030.248,453.311,341.637,176.720,49.176,160.514
C05213=1030.283,453.556,341.602,176.742,49.178,160.518
C05214=1030.327,453.861,341.558,176.769,49.182,160.523
C05215=1030.048,453.933,341.224,176.773,49.244,160.543
C05216=1030.010,453.669,341.261,176.749,49.241,160.539
C05217=1029.976,453.424,341.297,176.726,49.239,160.535
C05218=1029.941,453.178,341.333,176.705,49.236,160.530
C05219=1029.908,452.931,341.370,176.683,49.233,160.526
C05220=1029.874,452.687,341.406,176.662,49.231,160.522
C05221=1029.841,452.440,341.444,176.640,49.227,160.517
C05222=1029.809,452.195,341.482,176.618,49.224,160.513
C05223=1029.777,451.949,341.520,176.597,49.222,160.509
C05224=1029.746,451.704,341.559,176.575,49.219,160.504
C05225=1029.714,451.458,341.597,176.554,49.216,160.500
C05226=1029.684,451.212,341.637,176.533,49.213,160.496
C05227=1029.654,450.967,341.677,176.511,49.209,160.491
C05228=1029.624,450.722,341.717,176.490,49.206,160.487
C05229=1029.595,450.477,341.757,176.470,49.203,160.483
C05230=1029.566,450.231,341.798,176.449,49.199,160.478
C05231=1029.538,449.986,341.839,176.428,49.196,160.474
C05232=1029.510,449.740,341.881,176.408,49.192,160.470
C05233=1029.484,449.495,341.923,176.387,49.188,160.465
C05234=1029.457,449.250,341.966,176.366,49.185,160.461
C05235=1029.431,449.005,342.009,176.346,49.181,160.457
C05236=1029.405,448.759,342.052,176.325,49.178,160.452
C05237=1029.380,448.515,342.096,176.305,49.173,160.448
C05238=1029.356,448.270,342.140,176.286,49.170,160.444
C05239=1029.331,448.025,342.185,176.265,49.166,160.439
C05240=1029.307,447.780,342.230,176.245,49.161,160.435
C05241=1029.284,447.536,342.275,176.225,49.158,160.430
C05242=1029.261,447.291,342.321,176.205,49.153,160.426
C05243=1029.239,447.047,342.367,176.186,49.149,160.422
C05244=1029.217,446.802,342.415,176.166,49.145,160.417
C05245=1029.195,446.557,342.461,176.147,49.140,160.413
C05246=1029.175,446.314,342.509,176.127,49.136,160.408
C05247=1029.154,446.069,342.556,176.108,49.131,160.404
C05248=1029.134,445.825,342.604,176.089,49.127,160.400
C05249=1029.114,445.581,342.653,176.069,49.122,160.395
C05250=1029.095,445.337,342.703,176.050,49.117,160.391
C05251=1029.077,445.093,342.752,176.032,49.112,160.386
C05252=1029.058,444.849,342.802,176.013,49.108,160.382
C05253=1029.041,444.605,342.852,175.994,49.103,160.377
C05254=1029.024,444.362,342.902,175.974,49.097,160.373
C05255=1029.007,444.118,342.953,175.956,49.092,160.368
C05256=1028.991,443.873,343.005,175.938,49.087,160.364
C05257=1028.976,443.630,343.056,175.919,49.082,160.359
C05258=1028.960,443.387,343.109,175.900,49.077,160.355
C05259=1028.945,443.144,343.162,175.882,49.072,160.351
C05260=1028.932,442.901,343.215,175.864,49.066,160.346
C05261=1028.917,442.658,343.268,175.845,49.060,160.341
C05262=1028.903,442.413,343.321,175.827,49.055,160.337
C05263=1028.890,442.170,343.375,175.810,49.049,160.333
C05264=1028.876,441.926,343.428,175.792,49.043,160.328
C05265=1028.861,441.682,343.481,175.773,49.038,160.324
C05266=1028.848,441.438,343.534,175.755,49.033,160.319
C05267=1028.834,441.195,343.587,175.738,49.027,160.315
C05268=1028.820,440.950,343.641,175.720,49.022,160.311
C05269=1028.807,440.707,343.693,175.702,49.017,160.306
C05270=1028.793,440.463,343.746,175.685,49.011,160.302
C05271=1028.780,440.219,343.799,175.667,49.006,160.297
C05272=1028.764,439.947,343.857,175.648,49.000,160.293
C05273=1028.750,439.677,343.917,175.629,48.994,160.288
C05274=1028.734,439.405,343.975,175.609,48.988,160.283
C05275=1028.719,439.135,344.034,175.590,48.982,160.279
C05276=1028.706,438.890,344.086,175.572,48.977,160.274
C05277=1028.692,438.646,344.139,175.555,48.972,160.270
C05278=1028.680,438.402,344.191,175.538,48.966,160.266
C05279=1028.666,438.158,344.243,175.521,48.961,160.262
C05280=1028.652,437.914,344.296,175.504,48.956,160.257
C05281=1028.639,437.669,344.348,175.487,48.951,160.253
C05282=1028.626,437.425,344.400,175.470,48.946,160.249
C05283=1028.612,437.181,344.452,175.454,48.941,160.245
C05284=1028.600,436.936,344.504,175.437,48.936,160.241
C05285=1028.587,436.693,344.556,175.420,48.930,160.237
C05286=1028.573,436.448,344.608,175.403,48.925,160.233
C05287=1028.560,436.204,344.660,175.387,48.921,160.229
C05288=1028.547,435.959,344.712,175.370,48.915,160.225
C05289=1028.534,435.716,344.764,175.354,48.910,160.221
C05290=1028.520,435.472,344.816,175.337,48.906,160.217
C05291=1028.508,435.226,344.867,175.321,48.900,160.213
C05292=1028.495,434.983,344.919,175.304,48.896,160.209
C05293=1028.482,434.738,344.970,175.288,48.891,160.205
C05294=1028.469,434.494,345.022,175.272,48.886,160.201
C05295=1028.456,434.249,345.073,175.256,48.881,160.197
C05296=1028.443,434.005,345.125,175.240,48.876,160.193
C05297=1028.430,433.761,345.176,175.224,48.871,160.190
C05298=1028.418,433.516,345.227,175.208,48.866,160.186
C05299=1028.405,433.271,345.279,175.192,48.862,160.182
C05300=1028.393,433.027,345.329,175.176,48.857,160.178
C05301=1028.380,432.783,345.380,175.160,48.852,160.174
C05302=1028.367,432.538,345.431,175.145,48.848,160.171
C05303=1028.354,432.294,345.482,175.129,48.843,160.167
C05304=1028.341,432.049,345.533,175.113,48.838,160.163
C05305=1028.328,431.805,345.584,175.097,48.834,160.159
C05306=1028.316,431.560,345.635,175.082,48.828,160.155
C05307=1028.303,431.316,345.685,175.066,48.824,160.152
C05308=1028.291,431.071,345.736,175.051,48.820,160.148
C05309=1028.278,430.827,345.787,175.036,48.815,160.144
C05310=1028.266,430.582,345.837,175.021,48.810,160.141
C05311=1028.253,430.337,345.888,175.005,48.806,160.137
C05312=1028.240,430.093,345.938,174.990,48.801,160.134
C05313=1028.228,429.848,345.988,174.975,48.797,160.130
C05314=1028.215,429.604,346.039,174.960,48.792,160.126
C05315=1028.203,429.359,346.089,174.945,48.788,160.123
C05316=1028.191,429.115,346.139,174.929,48.783,160.119
C05317=1028.179,428.870,346.190,174.914,48.779,160.116
C05318=1028.166,428.626,346.240,174.899,48.774,160.112
C05319=1028.154,428.381,346.290,174.884,48.770,160.109
C05320=1028.137,428.027,346.362,174.863,48.764,160.104
C05321=1028.120,427.673,346.434,174.841,48.757,160.099
C05322=1028.102,427.320,346.506,174.820,48.751,160.093
C05323=1028.085,426.966,346.578,174.799,48.745,160.089
C05324=1028.072,426.721,346.628,174.785,48.740,160.085
C05325=1028.061,426.477,346.678,174.770,48.736,160.082
C05326=1028.049,426.232,346.727,174.755,48.732,160.078
C05327=1028.036,425.987,346.778,174.742,48.727,160.075
C05328=1028.025,425.768,346.821,174.728,48.724,160.072
C05329=1028.015,425.549,346.866,174.715,48.720,160.069
C05330=1028.004,425.330,346.910,174.702,48.716,160.066
C05331=1027.993,425.110,346.954,174.690,48.712,160.063
C05332=1027.983,424.891,346.999,174.677,48.709,160.060
C05333=1027.972,424.672,347.042,174.664,48.705,160.057
C05334=1027.961,424.452,347.087,174.652,48.701,160.054
C05335=1027.951,424.232,347.131,174.639,48.698,160.051
C05336=1027.939,423.988,347.179,174.626,48.694,160.048
C05337=1027.927,423.743,347.228,174.611,48.690,160.045
C05338=1027.915,423.497,347.278,174.596,48.686,160.041
C05339=1027.904,423.253,347.327,174.583,48.682,160.038
C05340=1027.892,423.008,347.376,174.570,48.677,160.035
C05341=1027.880,422.764,347.424,174.555,48.674,160.032
C05342=1027.868,422.518,347.474,174.542,48.669,160.028
C05343=1027.857,422.273,347.522,174.528,48.666,160.025
C05344=1027.846,422.028,347.571,174.514,48.662,160.022
C05345=1027.834,421.784,347.619,174.500,48.658,160.019
C05346=1027.822,421.538,347.668,174.487,48.654,160.016
C05347=1027.810,421.293,347.716,174.473,48.650,160.013
C05348=1027.799,421.048,347.765,174.459,48.646,160.010
C05349=1027.787,420.803,347.814,174.446,48.642,160.007
C05350=1027.775,420.558,347.861,174.433,48.638,160.003
C05351=1027.764,420.313,347.910,174.419,48.634,160.000
C05352=1027.752,420.068,347.958,174.405,48.631,159.997
C05353=1027.741,419.823,348.006,174.392,48.627,159.994
C05354=1027.730,419.577,348.055,174.379,48.623,159.991
C05355=1027.718,419.332,348.102,174.366,48.619,159.988
C05356=1027.707,419.087,348.151,174.353,48.615,159.985
C05357=1027.695,418.842,348.198,174.340,48.612,159.982
C05358=1027.684,418.597,348.247,174.327,48.608,159.979
C05359=1027.673,418.352,348.294,174.314,48.605,159.976
C05360=1027.662,418.107,348.342,174.301,48.601,159.973
C05361=1027.651,417.862,348.391,174.288,48.597,159.971
C05362=1027.639,417.616,348.438,174.275,48.593,159.967
C05363=1027.628,417.372,348.486,174.262,48.590,159.965
C05364=1027.617,417.126,348.533,174.249,48.586,159.962
C05365=1027.606,416.881,348.582,174.236,48.583,159.959
C05366=1027.595,416.636,348.630,174.223,48.579,159.956
C05367=1027.584,416.390,348.677,174.210,48.576,159.953
C05368=1027.573,416.145,348.725,174.197,48.572,159.950
C05369=1027.562,415.900,348.771,174.184,48.569,159.947
C05370=1027.550,415.655,348.819,174.171,48.565,159.944
C05371=1027.539,415.409,348.867,174.160,48.562,159.942
C05372=1027.528,415.164,348.913,174.147,48.558,159.939
C05373=1027.517,414.918,348.960,174.134,48.555,159.936
C05374=1027.506,414.674,349.008,174.121,48.551,159.933
C05375=1027.495,414.428,349.055,174.108,48.548,159.930
C05376=1027.484,414.183,349.102,174.097,48.545,159.928
C05377=1027.473,413.937,349.149,174.084,48.541,159.925
C05378=1027.462,413.692,349.196,174.071,48.538,159.922
C05379=1027.450,413.446,349.243,174.060,48.535,159.919
C05380=1027.440,413.201,349.290,174.047,48.531,159.917
C05381=1027.429,412.956,349.337,174.034,48.528,159.914
C05382=1027.418,412.711,349.384,174.022,48.524,159.911
C05383=1027.407,412.465,349.431,174.010,48.522,159.908
C05384=1027.397,412.220,349.477,173.998,48.518,159.906
C05385=1027.386,411.975,349.524,173.986,48.515,159.903
C05386=1027.376,411.729,349.571,173.974,48.512,159.900
C05387=1027.364,411.484,349.618,173.962,48.509,159.898
C05388=1027.354,411.238,349.664,173.950,48.505,159.895
C05389=1027.343,410.993,349.711,173.937,48.502,159.892
C05390=1027.333,410.747,349.757,173.926,48.499,159.890
C05391=1027.322,410.502,349.803,173.913,48.496,159.887
C05392=1027.309,410.210,349.859,173.899,48.492,159.884
C05393=1027.297,409.918,349.914,173.885,48.488,159.881
C05394=1027.284,409.626,349.969,173.871,48.484,159.878
C05395=1027.271,409.334,350.024,173.857,48.481,159.875
C05396=1027.261,409.088,350.070,173.846,48.478,159.872
C05397=1027.250,408.842,350.116,173.834,48.475,159.870
C05398=1027.240,408.597,350.162,173.822,48.472,159.867
C05399=1027.229,408.351,350.208,173.810,48.469,159.865
C05400=1027.218,408.106,350.254,173.799,48.466,159.862
C05401=1027.208,407.860,350.300,173.788,48.463,159.860
C05402=1027.197,407.615,350.345,173.775,48.460,159.857
C05403=1027.186,407.370,350.390,173.764,48.458,159.855
C05404=1027.176,407.124,350.436,173.753,48.454,159.852
C05405=1027.165,406.879,350.482,173.742,48.452,159.850
C05406=1027.155,406.632,350.527,173.729,48.449,159.847
C05407=1027.145,406.387,350.573,173.718,48.446,159.845
C05408=1027.134,406.142,350.619,173.707,48.443,159.843
C05409=1027.123,405.896,350.665,173.696,48.440,159.840
C05410=1027.113,405.650,350.710,173.684,48.437,159.838
C05411=1027.103,405.405,350.756,173.673,48.434,159.835
C05412=1027.093,405.159,350.801,173.662,48.432,159.833
C05413=1027.083,404.914,350.846,173.651,48.429,159.831
C05414=1027.072,404.668,350.891,173.640,48.426,159.828
C05415=1027.062,404.422,350.937,173.629,48.423,159.826
C05416=1027.052,404.177,350.982,173.618,48.421,159.824
C05417=1027.042,403.931,351.028,173.607,48.418,159.821
C05418=1027.032,403.686,351.073,173.595,48.415,159.819
C05419=1027.021,403.439,351.118,173.584,48.413,159.817
C05420=1027.012,403.194,351.163,173.573,48.410,159.814
C05421=1027.002,402.949,351.208,173.562,48.407,159.812
C05422=1026.991,402.703,351.254,173.551,48.404,159.810
C05423=1026.982,402.457,351.298,173.540,48.402,159.807
C05424=1026.972,402.212,351.343,173.529,48.399,159.805
C05425=1026.962,401.966,351.388,173.518,48.397,159.803
C05426=1026.952,401.720,351.433,173.508,48.394,159.801
C05427=1026.942,401.475,351.478,173.497,48.391,159.798
C05428=1026.931,401.229,351.523,173.486,48.389,159.796
C05429=1026.921,400.983,351.568,173.475,48.386,159.794
C05430=1026.912,400.738,351.612,173.465,48.384,159.792
C05431=1026.902,400.492,351.657,173.453,48.381,159.789
C05432=1026.892,400.246,351.702,173.444,48.379,159.787
C05433=1026.882,400.000,351.746,173.433,48.376,159.785
C05434=1026.872,399.755,351.791,173.422,48.374,159.783
C05435=1026.862,399.509,351.836,173.411,48.372,159.781
C05436=1026.853,399.263,351.880,173.401,48.369,159.778
C05437=1026.842,399.018,351.924,173.390,48.367,159.776
C05438=1026.833,398.772,351.968,173.379,48.364,159.774
C05439=1026.823,398.525,352.013,173.370,48.362,159.772
C05440=1026.812,398.280,352.057,173.359,48.360,159.770
C05441=1026.803,398.034,352.102,173.348,48.357,159.768
C05442=1026.793,397.788,352.145,173.338,48.355,159.765
C05443=1026.783,397.542,352.189,173.328,48.353,159.763
C05444=1026.774,397.296,352.233,173.317,48.350,159.761
C05445=1026.763,397.051,352.277,173.307,48.348,159.759
C05446=1026.754,396.805,352.322,173.296,48.346,159.757
C05447=1026.744,396.559,352.365,173.287,48.343,159.755
C05448=1026.734,396.313,352.409,173.276,48.342,159.753
C05449=1026.724,396.067,352.453,173.266,48.339,159.751
C05450=1026.715,395.821,352.496,173.256,48.337,159.749
C05451=1026.705,395.576,352.540,173.246,48.334,159.747
C05452=1026.695,395.306,352.588,173.234,48.332,159.744
C05453=1026.684,395.034,352.637,173.223,48.330,159.742
C05454=1026.674,394.765,352.685,173.212,48.327,159.740
C05455=1026.663,394.495,352.733,173.202,48.325,159.738
